Yaskawa INFORM job: DEMO_ROOF_UPPER_0625_3PAINT_4.JBI

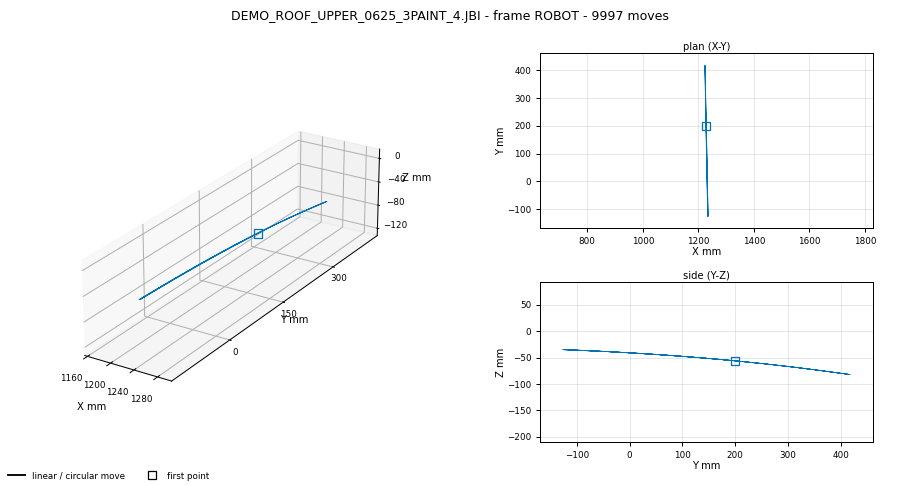
[picture p0: tool path of DEMO_ROOF_UPPER_0625_3PAINT_4.JBI in frame ROBOT, 9997 of 9997 moves have a stored position in this frame; points joined in program order, loops and branches not executed]
/JOB
//NAME DEMO_ROOF_UPPER_0625_3PAINT4
//POS
///NPOS 9997,0,0,0,0,0
///TOOL 0
///USER 0
///POSTYPE ROBOT
///RECTAN
///RCONF 1,0,0,0,0,0,0,0,0,0,0,0,0,0,0,0,0,0,0,0,0,0,0,0
C00000=1228.905,199.676,-56.077,-177.389,5.994,148.293
C00001=1228.909,199.428,-56.053,-177.392,5.993,148.294
C00002=1228.914,199.179,-56.029,-177.394,5.992,148.294
C00003=1228.919,198.930,-56.005,-177.396,5.990,148.294
C00004=1228.923,198.681,-55.981,-177.400,5.988,148.295
C00005=1228.928,198.432,-55.958,-177.402,5.986,148.295
C00006=1228.933,198.184,-55.934,-177.404,5.985,148.296
C00007=1228.937,197.935,-55.911,-177.407,5.983,148.296
C00008=1228.942,197.686,-55.887,-177.410,5.982,148.296
C00009=1228.946,197.437,-55.863,-177.412,5.980,148.297
C00010=1228.951,197.188,-55.840,-177.414,5.979,148.297
C00011=1228.956,196.939,-55.816,-177.417,5.977,148.298
C00012=1228.960,196.691,-55.792,-177.420,5.975,148.298
C00013=1228.965,196.442,-55.769,-177.423,5.973,148.298
C00014=1228.970,196.193,-55.746,-177.425,5.972,148.299
C00015=1228.974,195.944,-55.722,-177.427,5.971,148.299
C00016=1228.979,195.695,-55.698,-177.430,5.969,148.299
C00017=1228.983,195.446,-55.675,-177.433,5.968,148.300
C00018=1228.988,195.197,-55.652,-177.435,5.966,148.300
C00019=1228.992,194.949,-55.627,-177.438,5.964,148.301
C00020=1228.996,194.700,-55.605,-177.441,5.963,148.301
C00021=1229.001,194.451,-55.581,-177.443,5.961,148.301
C00022=1229.006,194.202,-55.558,-177.445,5.960,148.302
C00023=1229.010,193.953,-55.534,-177.448,5.958,148.302
C00024=1229.015,193.704,-55.511,-177.450,5.957,148.303
C00025=1229.020,193.455,-55.487,-177.453,5.955,148.303
C00026=1229.024,193.206,-55.464,-177.456,5.953,148.303
C00027=1229.029,192.957,-55.440,-177.458,5.952,148.304
C00028=1229.034,192.708,-55.417,-177.460,5.951,148.304
C00029=1229.039,192.461,-55.393,-177.464,5.949,148.305
C00030=1229.043,192.212,-55.371,-177.466,5.947,148.305
C00031=1229.047,191.963,-55.347,-177.468,5.946,148.305
C00032=1229.052,191.714,-55.324,-177.471,5.944,148.306
C00033=1229.057,191.465,-55.301,-177.474,5.942,148.306
C00034=1229.061,191.216,-55.277,-177.476,5.941,148.307
C00035=1229.066,190.967,-55.254,-177.479,5.940,148.307
C00036=1229.071,190.718,-55.231,-177.481,5.938,148.307
C00037=1229.075,190.469,-55.208,-177.484,5.937,148.308
C00038=1229.080,190.220,-55.184,-177.486,5.935,148.308
C00039=1229.084,189.971,-55.161,-177.489,5.933,148.308
C00040=1229.090,189.723,-55.138,-177.491,5.933,148.309
C00041=1229.094,189.474,-55.115,-177.494,5.931,148.309
C00042=1229.098,189.225,-55.092,-177.497,5.929,148.310
C00043=1229.103,188.976,-55.069,-177.499,5.928,148.310
C00044=1229.108,188.727,-55.045,-177.501,5.926,148.311
C00045=1229.112,188.478,-55.022,-177.505,5.925,148.311
C00046=1229.116,188.229,-54.999,-177.507,5.924,148.311
C00047=1229.121,187.980,-54.976,-177.509,5.922,148.312
C00048=1229.126,187.732,-54.953,-177.512,5.920,148.312
C00049=1229.131,187.483,-54.929,-177.514,5.919,148.313
C00050=1229.135,187.234,-54.907,-177.517,5.917,148.313
C00051=1229.140,186.985,-54.883,-177.520,5.916,148.313
C00052=1229.144,186.736,-54.860,-177.522,5.915,148.314
C00053=1229.149,186.487,-54.837,-177.525,5.913,148.314
C00054=1229.153,186.238,-54.814,-177.527,5.911,148.315
C00055=1229.158,185.968,-54.789,-177.530,5.909,148.315
C00056=1229.164,185.699,-54.764,-177.533,5.907,148.315
C00057=1229.168,185.429,-54.739,-177.536,5.907,148.316
C00058=1229.174,185.159,-54.714,-177.538,5.905,148.316
C00059=1229.178,184.910,-54.691,-177.541,5.903,148.317
C00060=1229.183,184.662,-54.668,-177.544,5.902,148.317
C00061=1229.187,184.413,-54.645,-177.546,5.901,148.318
C00062=1229.192,184.164,-54.622,-177.549,5.899,148.318
C00063=1229.196,183.915,-54.600,-177.551,5.898,148.318
C00064=1229.201,183.666,-54.576,-177.553,5.896,148.319
C00065=1229.206,183.418,-54.554,-177.557,5.894,148.319
C00066=1229.211,183.168,-54.531,-177.559,5.893,148.320
C00067=1229.215,182.919,-54.508,-177.561,5.892,148.320
C00068=1229.219,182.670,-54.485,-177.564,5.890,148.320
C00069=1229.225,182.422,-54.462,-177.567,5.889,148.321
C00070=1229.229,182.173,-54.440,-177.569,5.887,148.321
C00071=1229.234,181.924,-54.417,-177.572,5.885,148.322
C00072=1229.238,181.675,-54.393,-177.574,5.884,148.322
C00073=1229.242,181.426,-54.371,-177.577,5.883,148.323
C00074=1229.248,181.177,-54.348,-177.579,5.882,148.323
C00075=1229.252,180.928,-54.326,-177.582,5.880,148.323
C00076=1229.257,180.679,-54.302,-177.584,5.878,148.324
C00077=1229.261,180.431,-54.281,-177.587,5.877,148.324
C00078=1229.266,180.182,-54.257,-177.590,5.876,148.325
C00079=1229.270,179.932,-54.235,-177.592,5.874,148.325
C00080=1229.275,179.683,-54.212,-177.594,5.873,148.326
C00081=1229.280,179.435,-54.189,-177.598,5.871,148.326
C00082=1229.285,179.186,-54.167,-177.600,5.870,148.327
C00083=1229.289,178.936,-54.143,-177.602,5.868,148.327
C00084=1229.294,178.687,-54.121,-177.605,5.867,148.327
C00085=1229.299,178.439,-54.098,-177.608,5.866,148.328
C00086=1229.303,178.190,-54.076,-177.610,5.864,148.328
C00087=1229.307,177.941,-54.054,-177.612,5.863,148.329
C00088=1229.312,177.692,-54.031,-177.615,5.861,148.329
C00089=1229.317,177.443,-54.008,-177.618,5.860,148.329
C00090=1229.321,177.194,-53.985,-177.620,5.859,148.330
C00091=1229.326,176.945,-53.963,-177.623,5.857,148.330
C00092=1229.331,176.696,-53.940,-177.625,5.856,148.331
C00093=1229.335,176.447,-53.918,-177.628,5.854,148.331
C00094=1229.341,176.199,-53.895,-177.631,5.852,148.332
C00095=1229.345,175.949,-53.873,-177.633,5.851,148.332
C00096=1229.349,175.701,-53.850,-177.636,5.850,148.333
C00097=1229.354,175.452,-53.828,-177.638,5.849,148.333
C00098=1229.359,175.202,-53.806,-177.641,5.847,148.333
C00099=1229.363,174.953,-53.783,-177.643,5.845,148.334
C00100=1229.368,174.705,-53.761,-177.646,5.845,148.334
C00101=1229.372,174.456,-53.738,-177.649,5.843,148.335
C00102=1229.378,174.207,-53.716,-177.651,5.842,148.335
C00103=1229.382,173.958,-53.693,-177.654,5.840,148.336
C00104=1229.387,173.709,-53.670,-177.656,5.839,148.336
C00105=1229.392,173.460,-53.649,-177.658,5.837,148.336
C00106=1229.396,173.211,-53.626,-177.661,5.836,148.337
C00107=1229.401,172.962,-53.603,-177.664,5.835,148.337
C00108=1229.405,172.713,-53.582,-177.666,5.833,148.338
C00109=1229.409,172.464,-53.559,-177.668,5.832,148.338
C00110=1229.415,172.215,-53.537,-177.672,5.831,148.339
C00111=1229.419,171.966,-53.515,-177.674,5.830,148.339
C00112=1229.424,171.718,-53.492,-177.676,5.828,148.339
C00113=1229.428,171.469,-53.470,-177.679,5.826,148.340
C00114=1229.433,171.219,-53.447,-177.682,5.825,148.340
C00115=1229.438,170.970,-53.426,-177.684,5.823,148.341
C00116=1229.442,170.722,-53.403,-177.686,5.822,148.341
C00117=1229.448,170.473,-53.381,-177.689,5.821,148.342
C00118=1229.452,170.223,-53.359,-177.692,5.820,148.342
C00119=1229.457,169.975,-53.337,-177.694,5.818,148.342
C00120=1229.461,169.726,-53.314,-177.697,5.817,148.343
C00121=1229.466,169.476,-53.292,-177.699,5.816,148.343
C00122=1229.471,169.228,-53.270,-177.702,5.814,148.344
C00123=1229.475,168.978,-53.248,-177.705,5.813,148.344
C00124=1229.480,168.730,-53.226,-177.707,5.811,148.345
C00125=1229.485,168.480,-53.204,-177.709,5.810,148.345
C00126=1229.489,168.232,-53.181,-177.713,5.809,148.346
C00127=1229.494,167.983,-53.159,-177.715,5.808,148.346
C00128=1229.498,167.734,-53.137,-177.717,5.806,148.346
C00129=1229.503,167.485,-53.115,-177.720,5.805,148.347
C00130=1229.508,167.236,-53.093,-177.723,5.803,148.347
C00131=1229.513,166.986,-53.071,-177.725,5.802,148.348
C00132=1229.517,166.738,-53.049,-177.728,5.801,148.348
C00133=1229.522,166.488,-53.027,-177.730,5.800,148.349
C00134=1229.526,166.240,-53.005,-177.733,5.798,148.349
C00135=1229.531,165.991,-52.983,-177.736,5.797,148.350
C00136=1229.536,165.742,-52.961,-177.738,5.796,148.350
C00137=1229.540,165.493,-52.939,-177.740,5.794,148.350
C00138=1229.545,165.244,-52.917,-177.743,5.793,148.351
C00139=1229.550,164.995,-52.895,-177.746,5.791,148.351
C00140=1229.554,164.746,-52.873,-177.748,5.790,148.352
C00141=1229.559,164.497,-52.851,-177.751,5.789,148.352
C00142=1229.564,164.248,-52.829,-177.753,5.788,148.353
C00143=1229.568,163.999,-52.807,-177.756,5.786,148.353
C00144=1229.573,163.750,-52.786,-177.758,5.785,148.354
C00145=1229.578,163.501,-52.763,-177.761,5.783,148.354
C00146=1229.583,163.252,-52.741,-177.763,5.782,148.355
C00147=1229.587,163.003,-52.720,-177.766,5.781,148.355
C00148=1229.592,162.754,-52.698,-177.768,5.780,148.356
C00149=1229.597,162.505,-52.676,-177.771,5.778,148.356
C00150=1229.601,162.256,-52.654,-177.774,5.777,148.357
C00151=1229.606,162.007,-52.633,-177.776,5.776,148.357
C00152=1229.611,161.758,-52.611,-177.779,5.775,148.358
C00153=1229.615,161.509,-52.589,-177.781,5.773,148.358
C00154=1229.620,161.260,-52.568,-177.784,5.772,148.358
C00155=1229.624,161.011,-52.545,-177.787,5.771,148.359
C00156=1229.629,160.762,-52.524,-177.789,5.770,148.359
C00157=1229.634,160.513,-52.502,-177.791,5.768,148.360
C00158=1229.638,160.264,-52.480,-177.794,5.767,148.360
C00159=1229.644,159.995,-52.457,-177.797,5.765,148.361
C00160=1229.649,159.726,-52.434,-177.800,5.764,148.361
C00161=1229.654,159.457,-52.410,-177.802,5.763,148.362
C00162=1229.659,159.188,-52.386,-177.805,5.761,148.362
C00163=1229.663,158.938,-52.364,-177.807,5.760,148.363
C00164=1229.668,158.690,-52.343,-177.810,5.759,148.363
C00165=1229.673,158.441,-52.322,-177.812,5.758,148.364
C00166=1229.677,158.191,-52.300,-177.816,5.756,148.364
C00167=1229.682,157.943,-52.279,-177.818,5.755,148.365
C00168=1229.687,157.694,-52.257,-177.820,5.753,148.365
C00169=1229.691,157.444,-52.236,-177.823,5.753,148.366
C00170=1229.696,157.195,-52.214,-177.826,5.751,148.366
C00171=1229.701,156.947,-52.192,-177.828,5.750,148.366
C00172=1229.706,156.697,-52.171,-177.831,5.749,148.367
C00173=1229.711,156.448,-52.149,-177.833,5.748,148.367
C00174=1229.715,156.200,-52.128,-177.836,5.746,148.368
C00175=1229.720,155.950,-52.106,-177.838,5.745,148.368
C00176=1229.725,155.701,-52.085,-177.841,5.743,148.369
C00177=1229.729,155.453,-52.063,-177.843,5.743,148.369
C00178=1229.734,155.203,-52.042,-177.846,5.741,148.370
C00179=1229.738,154.954,-52.020,-177.849,5.740,148.370
C00180=1229.743,154.705,-51.999,-177.851,5.739,148.371
C00181=1229.748,154.456,-51.978,-177.853,5.737,148.371
C00182=1229.753,154.207,-51.956,-177.856,5.737,148.372
C00183=1229.757,153.958,-51.935,-177.859,5.735,148.372
C00184=1229.762,153.709,-51.914,-177.861,5.734,148.373
C00185=1229.766,153.460,-51.892,-177.864,5.732,148.373
C00186=1229.771,153.211,-51.871,-177.866,5.731,148.373
C00187=1229.776,152.962,-51.849,-177.869,5.730,148.374
C00188=1229.782,152.713,-51.828,-177.871,5.729,148.374
C00189=1229.785,152.464,-51.807,-177.874,5.727,148.375
C00190=1229.790,152.214,-51.786,-177.877,5.726,148.375
C00191=1229.795,151.966,-51.764,-177.879,5.726,148.376
C00192=1229.800,151.716,-51.743,-177.882,5.724,148.376
C00193=1229.804,151.467,-51.722,-177.884,5.723,148.377
C00194=1229.809,151.218,-51.701,-177.887,5.721,148.377
C00195=1229.814,150.970,-51.679,-177.889,5.720,148.378
C00196=1229.819,150.720,-51.658,-177.892,5.719,148.378
C00197=1229.823,150.471,-51.636,-177.894,5.718,148.379
C00198=1229.828,150.222,-51.615,-177.897,5.717,148.379
C00199=1229.833,149.973,-51.594,-177.900,5.715,148.380
C00200=1229.838,149.724,-51.573,-177.902,5.714,148.380
C00201=1229.842,149.476,-51.552,-177.905,5.713,148.381
C00202=1229.846,149.226,-51.530,-177.907,5.712,148.381
C00203=1229.852,148.977,-51.509,-177.910,5.710,148.382
C00204=1229.856,148.728,-51.488,-177.912,5.710,148.382
C00205=1229.861,148.479,-51.467,-177.915,5.709,148.383
C00206=1229.866,148.230,-51.446,-177.918,5.707,148.383
C00207=1229.870,147.980,-51.424,-177.920,5.706,148.384
C00208=1229.875,147.731,-51.404,-177.923,5.705,148.384
C00209=1229.880,147.483,-51.382,-177.925,5.704,148.385
C00210=1229.885,147.233,-51.361,-177.928,5.702,148.385
C00211=1229.889,146.985,-51.341,-177.930,5.701,148.386
C00212=1229.894,146.736,-51.319,-177.933,5.700,148.386
C00213=1229.898,146.486,-51.299,-177.935,5.699,148.387
C00214=1229.903,146.237,-51.278,-177.938,5.698,148.387
C00215=1229.908,145.988,-51.256,-177.941,5.696,148.388
C00216=1229.912,145.739,-51.236,-177.943,5.695,148.388
C00217=1229.918,145.490,-51.215,-177.945,5.695,148.389
C00218=1229.923,145.241,-51.194,-177.948,5.693,148.389
C00219=1229.926,144.992,-51.172,-177.951,5.692,148.390
C00220=1229.932,144.743,-51.151,-177.953,5.690,148.390
C00221=1229.936,144.494,-51.131,-177.956,5.690,148.391
C00222=1229.941,144.244,-51.110,-177.958,5.689,148.391
C00223=1229.945,143.996,-51.089,-177.961,5.687,148.392
C00224=1229.950,143.747,-51.068,-177.963,5.686,148.392
C00225=1229.956,143.498,-51.047,-177.967,5.685,148.393
C00226=1229.960,143.249,-51.026,-177.969,5.684,148.393
C00227=1229.965,142.999,-51.005,-177.971,5.683,148.394
C00228=1229.969,142.750,-50.985,-177.974,5.681,148.394
C00229=1229.974,142.501,-50.963,-177.976,5.681,148.395
C00230=1229.978,142.252,-50.943,-177.979,5.680,148.395
C00231=1229.984,142.003,-50.922,-177.981,5.678,148.395
C00232=1229.988,141.754,-50.901,-177.984,5.677,148.396
C00233=1229.993,141.505,-50.880,-177.987,5.675,148.396
C00234=1229.998,141.256,-50.860,-177.989,5.675,148.397
C00235=1230.003,141.006,-50.839,-177.991,5.674,148.397
C00236=1230.007,140.757,-50.819,-177.994,5.672,148.398
C00237=1230.012,140.509,-50.797,-177.997,5.671,148.398
C00238=1230.017,140.260,-50.777,-177.999,5.671,148.399
C00239=1230.021,140.010,-50.755,-178.002,5.669,148.399
C00240=1230.026,139.761,-50.735,-178.004,5.668,148.400
C00241=1230.031,139.512,-50.714,-178.007,5.666,148.400
C00242=1230.035,139.263,-50.694,-178.010,5.666,148.401
C00243=1230.040,139.014,-50.673,-178.012,5.665,148.401
C00244=1230.045,138.765,-50.652,-178.015,5.663,148.402
C00245=1230.049,138.516,-50.632,-178.017,5.662,148.403
C00246=1230.054,138.266,-50.611,-178.020,5.662,148.403
C00247=1230.059,138.017,-50.591,-178.022,5.660,148.404
C00248=1230.064,137.768,-50.570,-178.025,5.659,148.404
C00249=1230.068,137.519,-50.549,-178.027,5.658,148.405
C00250=1230.073,137.270,-50.529,-178.030,5.657,148.405
C00251=1230.078,137.021,-50.508,-178.032,5.656,148.406
C00252=1230.082,136.772,-50.487,-178.035,5.654,148.406
C00253=1230.087,136.523,-50.467,-178.038,5.653,148.407
C00254=1230.092,136.273,-50.447,-178.040,5.653,148.407
C00255=1230.097,136.024,-50.426,-178.043,5.651,148.408
C00256=1230.102,135.775,-50.406,-178.045,5.650,148.408
C00257=1230.106,135.526,-50.385,-178.048,5.649,148.409
C00258=1230.111,135.277,-50.365,-178.051,5.648,148.409
C00259=1230.116,135.028,-50.344,-178.053,5.647,148.410
C00260=1230.121,134.779,-50.323,-178.055,5.646,148.410
C00261=1230.125,134.530,-50.303,-178.058,5.644,148.411
C00262=1230.130,134.280,-50.283,-178.061,5.644,148.411
C00263=1230.135,134.012,-50.261,-178.063,5.643,148.412
C00264=1230.140,133.744,-50.239,-178.066,5.641,148.412
C00265=1230.146,133.475,-50.217,-178.069,5.640,148.413
C00266=1230.150,133.206,-50.195,-178.072,5.639,148.414
C00267=1230.155,132.957,-50.174,-178.074,5.638,148.414
C00268=1230.160,132.707,-50.154,-178.077,5.637,148.415
C00269=1230.165,132.459,-50.134,-178.079,5.636,148.415
C00270=1230.170,132.210,-50.113,-178.082,5.635,148.416
C00271=1230.175,131.961,-50.093,-178.084,5.633,148.416
C00272=1230.179,131.711,-50.073,-178.087,5.632,148.417
C00273=1230.184,131.462,-50.053,-178.089,5.631,148.417
C00274=1230.189,131.213,-50.032,-178.092,5.630,148.418
C00275=1230.193,130.964,-50.011,-178.095,5.629,148.418
C00276=1230.198,130.714,-49.992,-178.097,5.628,148.419
C00277=1230.203,130.465,-49.971,-178.100,5.627,148.419
C00278=1230.207,130.217,-49.951,-178.102,5.626,148.420
C00279=1230.212,129.967,-49.931,-178.105,5.625,148.420
C00280=1230.218,129.718,-49.911,-178.107,5.624,148.421
C00281=1230.222,129.469,-49.890,-178.110,5.623,148.421
C00282=1230.227,129.220,-49.871,-178.112,5.622,148.422
C00283=1230.231,128.971,-49.850,-178.115,5.621,148.422
C00284=1230.236,128.722,-49.829,-178.118,5.619,148.423
C00285=1230.241,128.472,-49.810,-178.120,5.619,148.423
C00286=1230.246,128.223,-49.789,-178.123,5.618,148.424
C00287=1230.250,127.974,-49.770,-178.125,5.616,148.424
C00288=1230.255,127.725,-49.750,-178.128,5.616,148.425
C00289=1230.260,127.476,-49.729,-178.130,5.615,148.425
C00290=1230.265,127.226,-49.709,-178.133,5.613,148.426
C00291=1230.270,126.978,-49.689,-178.135,5.612,148.426
C00292=1230.274,126.728,-49.669,-178.138,5.612,148.427
C00293=1230.279,126.479,-49.649,-178.140,5.611,148.428
C00294=1230.284,126.230,-49.629,-178.143,5.609,148.428
C00295=1230.289,125.981,-49.609,-178.146,5.609,148.429
C00296=1230.293,125.732,-49.589,-178.148,5.608,148.429
C00297=1230.298,125.483,-49.569,-178.151,5.606,148.430
C00298=1230.302,125.234,-49.549,-178.153,5.605,148.430
C00299=1230.307,124.984,-49.529,-178.156,5.605,148.431
C00300=1230.313,124.736,-49.508,-178.158,5.604,148.431
C00301=1230.317,124.486,-49.489,-178.161,5.602,148.432
C00302=1230.322,124.236,-49.469,-178.164,5.601,148.432
C00303=1230.327,123.988,-49.449,-178.166,5.600,148.433
C00304=1230.331,123.738,-49.429,-178.169,5.599,148.434
C00305=1230.336,123.490,-49.409,-178.171,5.598,148.434
C00306=1230.341,123.240,-49.389,-178.174,5.597,148.435
C00307=1230.346,122.991,-49.369,-178.176,5.596,148.435
C00308=1230.350,122.742,-49.349,-178.179,5.595,148.436
C00309=1230.355,122.493,-49.329,-178.182,5.594,148.436
C00310=1230.360,122.244,-49.310,-178.184,5.593,148.437
C00311=1230.365,121.994,-49.290,-178.186,5.593,148.437
C00312=1230.369,121.745,-49.270,-178.189,5.591,148.438
C00313=1230.374,121.496,-49.250,-178.192,5.590,148.438
C00314=1230.379,121.247,-49.231,-178.194,5.590,148.439
C00315=1230.384,120.998,-49.210,-178.196,5.589,148.439
C00316=1230.389,120.748,-49.191,-178.200,5.587,148.440
C00317=1230.393,120.499,-49.171,-178.202,5.586,148.440
C00318=1230.398,120.251,-49.151,-178.204,5.586,148.441
C00319=1230.403,120.001,-49.131,-178.206,5.585,148.441
C00320=1230.408,119.751,-49.112,-178.210,5.583,148.442
C00321=1230.413,119.503,-49.092,-178.212,5.583,148.443
C00322=1230.418,119.254,-49.072,-178.214,5.582,148.443
C00323=1230.422,119.004,-49.053,-178.217,5.581,148.444
C00324=1230.426,118.755,-49.033,-178.220,5.579,148.444
C00325=1230.431,118.507,-49.013,-178.222,5.579,148.445
C00326=1230.436,118.257,-48.994,-178.225,5.578,148.445
C00327=1230.441,118.007,-48.974,-178.227,5.577,148.446
C00328=1230.446,117.759,-48.955,-178.230,5.575,148.446
C00329=1230.451,117.510,-48.934,-178.233,5.575,148.447
C00330=1230.455,117.260,-48.915,-178.235,5.574,148.447
C00331=1230.461,117.011,-48.895,-178.237,5.573,148.448
C00332=1230.466,116.762,-48.876,-178.240,5.571,148.449
C00333=1230.470,116.512,-48.857,-178.243,5.571,148.449
C00334=1230.474,116.263,-48.836,-178.245,5.570,148.450
C00335=1230.479,116.014,-48.817,-178.247,5.569,148.450
C00336=1230.484,115.765,-48.797,-178.251,5.568,148.451
C00337=1230.489,115.516,-48.778,-178.253,5.567,148.451
C00338=1230.494,115.266,-48.758,-178.255,5.566,148.452
C00339=1230.499,115.017,-48.739,-178.258,5.566,148.453
C00340=1230.503,114.768,-48.720,-178.261,5.564,148.453
C00341=1230.508,114.519,-48.700,-178.263,5.563,148.454
C00342=1230.513,114.270,-48.680,-178.266,5.563,148.454
C00343=1230.518,114.021,-48.661,-178.268,5.562,148.455
C00344=1230.523,113.771,-48.641,-178.271,5.561,148.455
C00345=1230.527,113.522,-48.622,-178.273,5.559,148.456
C00346=1230.532,113.273,-48.603,-178.276,5.559,148.456
C00347=1230.537,113.024,-48.583,-178.279,5.558,148.457
C00348=1230.542,112.775,-48.564,-178.281,5.557,148.457
C00349=1230.547,112.525,-48.544,-178.283,5.556,148.458
C00350=1230.551,112.276,-48.525,-178.286,5.555,148.459
C00351=1230.556,112.027,-48.506,-178.289,5.554,148.459
C00352=1230.561,111.778,-48.486,-178.291,5.553,148.460
C00353=1230.566,111.529,-48.467,-178.293,5.552,148.460
C00354=1230.570,111.279,-48.448,-178.296,5.551,148.461
C00355=1230.575,111.030,-48.428,-178.299,5.550,148.461
C00356=1230.580,110.781,-48.409,-178.301,5.549,148.462
C00357=1230.584,110.532,-48.390,-178.304,5.549,148.462
C00358=1230.590,110.283,-48.370,-178.306,5.548,148.463
C00359=1230.595,110.033,-48.351,-178.309,5.546,148.463
C00360=1230.599,109.784,-48.331,-178.312,5.546,148.464
C00361=1230.604,109.535,-48.312,-178.314,5.545,148.465
C00362=1230.609,109.286,-48.293,-178.316,5.544,148.465
C00363=1230.614,109.037,-48.274,-178.319,5.543,148.466
C00364=1230.618,108.788,-48.254,-178.322,5.542,148.466
C00365=1230.623,108.539,-48.235,-178.324,5.541,148.467
C00366=1230.628,108.288,-48.216,-178.327,5.540,148.467
C00367=1230.633,108.021,-48.196,-178.330,5.540,148.468
C00368=1230.638,107.752,-48.175,-178.333,5.538,148.469
C00369=1230.643,107.484,-48.154,-178.335,5.537,148.469
C00370=1230.649,107.215,-48.134,-178.338,5.537,148.470
C00371=1230.654,106.965,-48.114,-178.341,5.535,148.470
C00372=1230.658,106.717,-48.096,-178.343,5.535,148.471
C00373=1230.663,106.467,-48.076,-178.345,5.534,148.472
C00374=1230.668,106.218,-48.057,-178.348,5.533,148.472
C00375=1230.673,105.969,-48.038,-178.351,5.532,148.473
C00376=1230.678,105.720,-48.019,-178.353,5.531,148.473
C00377=1230.682,105.470,-48.000,-178.356,5.530,148.474
C00378=1230.687,105.222,-47.981,-178.359,5.529,148.474
C00379=1230.691,104.972,-47.962,-178.361,5.528,148.475
C00380=1230.697,104.723,-47.943,-178.363,5.528,148.476
C00381=1230.702,104.473,-47.923,-178.366,5.527,148.476
C00382=1230.706,104.225,-47.905,-178.368,5.526,148.477
C00383=1230.711,103.975,-47.885,-178.371,5.525,148.477
C00384=1230.716,103.726,-47.867,-178.374,5.524,148.478
C00385=1230.721,103.476,-47.847,-178.376,5.523,148.478
C00386=1230.725,103.228,-47.829,-178.379,5.523,148.479
C00387=1230.731,102.978,-47.810,-178.381,5.522,148.480
C00388=1230.735,102.729,-47.791,-178.383,5.521,148.480
C00389=1230.740,102.480,-47.772,-178.386,5.520,148.481
C00390=1230.745,102.230,-47.753,-178.389,5.519,148.481
C00391=1230.750,101.981,-47.734,-178.392,5.518,148.482
C00392=1230.754,101.732,-47.715,-178.394,5.517,148.482
C00393=1230.760,101.483,-47.696,-178.396,5.517,148.483
C00394=1230.764,101.233,-47.677,-178.399,5.516,148.484
C00395=1230.769,100.985,-47.658,-178.402,5.514,148.484
C00396=1230.774,100.735,-47.640,-178.404,5.514,148.485
C00397=1230.779,100.486,-47.620,-178.407,5.513,148.485
C00398=1230.783,100.237,-47.603,-178.409,5.512,148.486
C00399=1230.788,99.987,-47.583,-178.412,5.512,148.486
C00400=1230.793,99.739,-47.564,-178.414,5.511,148.487
C00401=1230.798,99.488,-47.545,-178.416,5.510,148.487
C00402=1230.802,99.240,-47.527,-178.420,5.509,148.488
C00403=1230.807,98.991,-47.509,-178.422,5.508,148.489
C00404=1230.812,98.741,-47.489,-178.425,5.507,148.489
C00405=1230.817,98.492,-47.471,-178.427,5.506,148.490
C00406=1230.822,98.243,-47.452,-178.430,5.506,148.490
C00407=1230.827,97.993,-47.433,-178.432,5.505,148.491
C00408=1230.832,97.744,-47.414,-178.434,5.504,148.492
C00409=1230.836,97.494,-47.396,-178.437,5.504,148.492
C00410=1230.841,97.246,-47.377,-178.440,5.502,148.493
C00411=1230.847,96.996,-47.358,-178.442,5.501,148.493
C00412=1230.851,96.747,-47.339,-178.445,5.501,148.494
C00413=1230.856,96.498,-47.321,-178.448,5.500,148.495
C00414=1230.861,96.249,-47.302,-178.450,5.499,148.495
C00415=1230.865,95.999,-47.284,-178.452,5.498,148.496
C00416=1230.871,95.750,-47.264,-178.455,5.498,148.496
C00417=1230.875,95.501,-47.246,-178.458,5.497,148.497
C00418=1230.880,95.251,-47.228,-178.460,5.495,148.497
C00419=1230.885,95.002,-47.209,-178.463,5.495,148.498
C00420=1230.890,94.753,-47.191,-178.465,5.494,148.499
C00421=1230.894,94.504,-47.172,-178.468,5.494,148.499
C00422=1230.900,94.254,-47.153,-178.470,5.493,148.500
C00423=1230.905,94.005,-47.135,-178.473,5.492,148.500
C00424=1230.909,93.756,-47.116,-178.475,5.491,148.501
C00425=1230.914,93.507,-47.098,-178.478,5.491,148.502
C00426=1230.919,93.257,-47.080,-178.481,5.489,148.502
C00427=1230.923,93.008,-47.061,-178.483,5.488,148.503
C00428=1230.928,92.759,-47.043,-178.486,5.488,148.503
C00429=1230.934,92.509,-47.024,-178.488,5.487,148.504
C00430=1230.938,92.260,-47.005,-178.491,5.486,148.504
C00431=1230.943,92.011,-46.987,-178.493,5.486,148.505
C00432=1230.948,91.762,-46.969,-178.496,5.485,148.506
C00433=1230.953,91.513,-46.950,-178.498,5.484,148.506
C00434=1230.957,91.263,-46.931,-178.501,5.483,148.507
C00435=1230.962,91.014,-46.913,-178.503,5.483,148.507
C00436=1230.967,90.765,-46.895,-178.507,5.481,148.508
C00437=1230.971,90.515,-46.876,-178.509,5.480,148.509
C00438=1230.977,90.266,-46.858,-178.511,5.480,148.509
C00439=1230.982,90.017,-46.840,-178.514,5.479,148.510
C00440=1230.987,89.768,-46.822,-178.517,5.479,148.510
C00441=1230.991,89.518,-46.803,-178.519,5.478,148.511
C00442=1230.996,89.269,-46.784,-178.521,5.477,148.512
C00443=1231.001,89.020,-46.766,-178.524,5.476,148.512
C00444=1231.006,88.771,-46.748,-178.527,5.476,148.513
C00445=1231.010,88.521,-46.730,-178.529,5.475,148.513
C00446=1231.015,88.272,-46.711,-178.531,5.474,148.514
C00447=1231.020,88.023,-46.693,-178.534,5.473,148.515
C00448=1231.025,87.773,-46.675,-178.537,5.472,148.515
C00449=1231.030,87.524,-46.657,-178.539,5.471,148.516
C00450=1231.035,87.274,-46.638,-178.542,5.471,148.516
C00451=1231.040,87.025,-46.620,-178.544,5.470,148.517
C00452=1231.045,86.776,-46.602,-178.547,5.469,148.518
C00453=1231.049,86.527,-46.584,-178.549,5.468,148.518
C00454=1231.054,86.278,-46.566,-178.552,5.468,148.519
C00455=1231.058,86.028,-46.547,-178.554,5.467,148.519
C00456=1231.064,85.779,-46.529,-178.557,5.467,148.520
C00457=1231.069,85.530,-46.511,-178.559,5.466,148.520
C00458=1231.074,85.281,-46.493,-178.562,5.465,148.521
C00459=1231.079,85.031,-46.475,-178.564,5.465,148.522
C00460=1231.083,84.782,-46.456,-178.568,5.463,148.522
C00461=1231.088,84.532,-46.438,-178.570,5.462,148.523
C00462=1231.093,84.283,-46.420,-178.572,5.462,148.523
C00463=1231.098,84.034,-46.402,-178.575,5.461,148.524
C00464=1231.103,83.785,-46.384,-178.578,5.460,148.525
C00465=1231.108,83.536,-46.366,-178.580,5.460,148.525
C00466=1231.112,83.286,-46.348,-178.582,5.459,148.526
C00467=1231.117,83.037,-46.330,-178.585,5.458,148.527
C00468=1231.122,82.787,-46.312,-178.588,5.458,148.527
C00469=1231.127,82.538,-46.294,-178.590,5.457,148.528
C00470=1231.132,82.289,-46.276,-178.592,5.456,148.528
C00471=1231.137,82.021,-46.256,-178.595,5.455,148.529
C00472=1231.142,81.752,-46.237,-178.598,5.454,148.530
C00473=1231.148,81.484,-46.217,-178.601,5.453,148.530
C00474=1231.153,81.215,-46.199,-178.603,5.453,148.531
C00475=1231.158,80.966,-46.181,-178.606,5.452,148.532
C00476=1231.163,80.717,-46.163,-178.609,5.452,148.532
C00477=1231.168,80.468,-46.145,-178.611,5.451,148.533
C00478=1231.172,80.218,-46.126,-178.614,5.450,148.533
C00479=1231.177,79.969,-46.108,-178.616,5.449,148.534
C00480=1231.182,79.719,-46.090,-178.619,5.449,148.535
C00481=1231.187,79.470,-46.072,-178.621,5.448,148.535
C00482=1231.192,79.221,-46.054,-178.624,5.448,148.536
C00483=1231.197,78.971,-46.037,-178.626,5.447,148.536
C00484=1231.202,78.722,-46.019,-178.629,5.446,148.537
C00485=1231.207,78.473,-46.001,-178.631,5.446,148.538
C00486=1231.211,78.224,-45.984,-178.634,5.445,148.538
C00487=1231.216,77.975,-45.966,-178.637,5.444,148.539
C00488=1231.221,77.725,-45.949,-178.639,5.443,148.539
C00489=1231.226,77.476,-45.931,-178.642,5.442,148.540
C00490=1231.230,77.226,-45.912,-178.645,5.441,148.541
C00491=1231.235,76.977,-45.894,-178.647,5.441,148.541
C00492=1231.240,76.728,-45.876,-178.650,5.440,148.542
C00493=1231.245,76.478,-45.859,-178.652,5.439,148.542
C00494=1231.250,76.229,-45.841,-178.655,5.439,148.543
C00495=1231.254,75.980,-45.824,-178.657,5.438,148.544
C00496=1231.259,75.731,-45.806,-178.660,5.437,148.544
C00497=1231.264,75.481,-45.788,-178.662,5.437,148.545
C00498=1231.269,75.232,-45.770,-178.665,5.436,148.545
C00499=1231.274,74.982,-45.753,-178.667,5.435,148.546
C00500=1231.279,74.733,-45.735,-178.670,5.435,148.547
C00501=1231.284,74.484,-45.717,-178.672,5.434,148.547
C00502=1231.289,74.235,-45.700,-178.675,5.434,148.548
C00503=1231.293,73.985,-45.682,-178.677,5.433,148.549
C00504=1231.299,73.736,-45.665,-178.680,5.432,148.549
C00505=1231.304,73.487,-45.647,-178.683,5.431,148.550
C00506=1231.309,73.237,-45.629,-178.685,5.431,148.551
C00507=1231.313,72.988,-45.612,-178.688,5.430,148.551
C00508=1231.318,72.739,-45.594,-178.690,5.430,148.552
C00509=1231.323,72.489,-45.577,-178.693,5.429,148.552
C00510=1231.328,72.240,-45.559,-178.695,5.428,148.553
C00511=1231.333,71.991,-45.541,-178.698,5.428,148.554
C00512=1231.337,71.741,-45.524,-178.700,5.427,148.554
C00513=1231.342,71.492,-45.506,-178.703,5.426,148.555
C00514=1231.348,71.242,-45.489,-178.705,5.425,148.555
C00515=1231.352,70.993,-45.471,-178.708,5.425,148.556
C00516=1231.357,70.744,-45.454,-178.710,5.424,148.557
C00517=1231.362,70.494,-45.436,-178.713,5.424,148.557
C00518=1231.367,70.245,-45.418,-178.716,5.423,148.558
C00519=1231.372,69.995,-45.401,-178.718,5.422,148.559
C00520=1231.376,69.746,-45.384,-178.720,5.422,148.559
C00521=1231.381,69.497,-45.366,-178.723,5.421,148.560
C00522=1231.387,69.248,-45.349,-178.726,5.420,148.560
C00523=1231.391,68.999,-45.332,-178.728,5.420,148.561
C00524=1231.396,68.749,-45.314,-178.731,5.419,148.562
C00525=1231.402,68.500,-45.297,-178.734,5.419,148.562
C00526=1231.406,68.250,-45.279,-178.736,5.418,148.563
C00527=1231.411,68.001,-45.262,-178.738,5.417,148.564
C00528=1231.416,67.752,-45.244,-178.741,5.416,148.564
C00529=1231.421,67.502,-45.227,-178.744,5.416,148.565
C00530=1231.425,67.253,-45.210,-178.746,5.415,148.565
C00531=1231.430,67.003,-45.192,-178.749,5.415,148.566
C00532=1231.436,66.754,-45.175,-178.751,5.414,148.567
C00533=1231.440,66.505,-45.158,-178.754,5.413,148.567
C00534=1231.446,66.256,-45.141,-178.756,5.413,148.568
C00535=1231.450,66.007,-45.123,-178.759,5.412,148.569
C00536=1231.455,65.757,-45.106,-178.762,5.411,148.569
C00537=1231.460,65.508,-45.088,-178.764,5.411,148.570
C00538=1231.464,65.258,-45.071,-178.767,5.410,148.571
C00539=1231.470,65.009,-45.054,-178.769,5.409,148.571
C00540=1231.475,64.759,-45.036,-178.772,5.409,148.572
C00541=1231.479,64.510,-45.020,-178.774,5.409,148.572
C00542=1231.485,64.261,-45.003,-178.776,5.408,148.573
C00543=1231.489,64.012,-44.985,-178.779,5.408,148.574
C00544=1231.494,63.762,-44.968,-178.782,5.407,148.574
C00545=1231.499,63.513,-44.951,-178.784,5.406,148.575
C00546=1231.504,63.263,-44.933,-178.786,5.406,148.575
C00547=1231.509,63.014,-44.916,-178.789,5.405,148.576
C00548=1231.513,62.764,-44.899,-178.792,5.404,148.577
C00549=1231.519,62.516,-44.882,-178.794,5.404,148.577
C00550=1231.523,62.266,-44.865,-178.797,5.403,148.578
C00551=1231.529,62.016,-44.848,-178.799,5.403,148.579
C00552=1231.533,61.767,-44.831,-178.802,5.402,148.579
C00553=1231.538,61.518,-44.813,-178.804,5.401,148.580
C00554=1231.542,61.268,-44.797,-178.807,5.401,148.581
C00555=1231.548,61.019,-44.780,-178.810,5.400,148.581
C00556=1231.553,60.770,-44.763,-178.812,5.399,148.582
C00557=1231.558,60.520,-44.746,-178.815,5.399,148.583
C00558=1231.562,60.271,-44.728,-178.817,5.398,148.583
C00559=1231.567,60.021,-44.711,-178.820,5.398,148.584
C00560=1231.572,59.772,-44.695,-178.822,5.397,148.584
C00561=1231.578,59.523,-44.678,-178.825,5.396,148.585
C00562=1231.582,59.273,-44.661,-178.827,5.396,148.586
C00563=1231.587,59.024,-44.643,-178.830,5.395,148.586
C00564=1231.592,58.775,-44.627,-178.832,5.395,148.587
C00565=1231.597,58.525,-44.609,-178.835,5.395,148.588
C00566=1231.602,58.276,-44.593,-178.837,5.394,148.588
C00567=1231.607,58.026,-44.575,-178.840,5.393,148.589
C00568=1231.612,57.777,-44.559,-178.842,5.393,148.589
C00569=1231.617,57.528,-44.542,-178.845,5.392,148.590
C00570=1231.621,57.279,-44.524,-178.847,5.391,148.591
C00571=1231.626,57.029,-44.508,-178.850,5.391,148.591
C00572=1231.631,56.779,-44.490,-178.853,5.390,148.592
C00573=1231.636,56.531,-44.474,-178.855,5.390,148.593
C00574=1231.641,56.281,-44.457,-178.858,5.389,148.593
C00575=1231.646,56.012,-44.439,-178.861,5.389,148.594
C00576=1231.652,55.744,-44.420,-178.863,5.388,148.595
C00577=1231.657,55.476,-44.402,-178.866,5.387,148.595
C00578=1231.662,55.208,-44.385,-178.869,5.387,148.596
C00579=1231.667,54.958,-44.367,-178.871,5.386,148.597
C00580=1231.672,54.708,-44.351,-178.874,5.386,148.597
C00581=1231.678,54.459,-44.334,-178.876,5.385,148.598
C00582=1231.682,54.210,-44.317,-178.879,5.385,148.599
C00583=1231.687,53.960,-44.300,-178.881,5.384,148.599
C00584=1231.692,53.711,-44.284,-178.884,5.383,148.600
C00585=1231.697,53.462,-44.267,-178.886,5.382,148.601
C00586=1231.701,53.212,-44.250,-178.889,5.383,148.601
C00587=1231.707,52.962,-44.233,-178.891,5.382,148.602
C00588=1231.712,52.714,-44.217,-178.894,5.382,148.603
C00589=1231.716,52.464,-44.201,-178.896,5.381,148.603
C00590=1231.722,52.214,-44.183,-178.899,5.380,148.604
C00591=1231.727,51.965,-44.167,-178.902,5.380,148.605
C00592=1231.731,51.716,-44.150,-178.904,5.379,148.605
C00593=1231.736,51.466,-44.134,-178.907,5.378,148.606
C00594=1231.741,51.217,-44.117,-178.909,5.378,148.606
C00595=1231.746,50.967,-44.100,-178.912,5.377,148.607
C00596=1231.750,50.718,-44.084,-178.914,5.377,148.608
C00597=1231.756,50.469,-44.067,-178.916,5.377,148.608
C00598=1231.761,50.219,-44.050,-178.919,5.376,148.609
C00599=1231.765,49.970,-44.033,-178.922,5.376,148.610
C00600=1231.771,49.721,-44.018,-178.924,5.375,148.610
C00601=1231.776,49.471,-44.000,-178.927,5.375,148.611
C00602=1231.781,49.222,-43.984,-178.929,5.374,148.611
C00603=1231.785,48.972,-43.968,-178.932,5.373,148.612
C00604=1231.790,48.723,-43.951,-178.934,5.372,148.613
C00605=1231.796,48.474,-43.934,-178.937,5.372,148.613
C00606=1231.800,48.224,-43.918,-178.940,5.371,148.614
C00607=1231.805,47.974,-43.901,-178.942,5.372,148.615
C00608=1231.810,47.726,-43.885,-178.944,5.371,148.615
C00609=1231.814,47.476,-43.868,-178.947,5.370,148.616
C00610=1231.820,47.227,-43.851,-178.950,5.370,148.617
C00611=1231.825,46.977,-43.835,-178.952,5.369,148.617
C00612=1231.830,46.727,-43.819,-178.955,5.369,148.618
C00613=1231.835,46.479,-43.803,-178.957,5.368,148.619
C00614=1231.839,46.229,-43.786,-178.960,5.367,148.619
C00615=1231.845,45.980,-43.770,-178.962,5.367,148.620
C00616=1231.850,45.730,-43.753,-178.964,5.367,148.621
C00617=1231.854,45.480,-43.736,-178.967,5.366,148.621
C00618=1231.860,45.231,-43.721,-178.970,5.366,148.622
C00619=1231.864,44.982,-43.704,-178.972,5.365,148.623
C00620=1231.869,44.733,-43.688,-178.975,5.365,148.623
C00621=1231.874,44.483,-43.671,-178.978,5.364,148.624
C00622=1231.879,44.234,-43.656,-178.980,5.364,148.625
C00623=1231.884,43.984,-43.638,-178.983,5.363,148.625
C00624=1231.889,43.735,-43.622,-178.985,5.363,148.626
C00625=1231.894,43.485,-43.606,-178.987,5.362,148.626
C00626=1231.899,43.236,-43.589,-178.990,5.362,148.627
C00627=1231.904,42.986,-43.574,-178.992,5.361,148.628
C00628=1231.908,42.737,-43.557,-178.995,5.361,148.628
C00629=1231.914,42.488,-43.541,-178.998,5.360,148.629
C00630=1231.918,42.238,-43.525,-179.000,5.359,148.630
C00631=1231.923,41.989,-43.509,-179.003,5.359,148.630
C00632=1231.928,41.740,-43.492,-179.005,5.359,148.631
C00633=1231.934,41.490,-43.476,-179.008,5.359,148.632
C00634=1231.938,41.240,-43.459,-179.010,5.358,148.633
C00635=1231.944,40.991,-43.443,-179.013,5.357,148.633
C00636=1231.948,40.742,-43.427,-179.016,5.357,148.634
C00637=1231.954,40.492,-43.411,-179.018,5.356,148.635
C00638=1231.958,40.243,-43.394,-179.021,5.356,148.635
C00639=1231.964,39.993,-43.379,-179.022,5.356,148.636
C00640=1231.968,39.744,-43.362,-179.025,5.355,148.636
C00641=1231.973,39.495,-43.346,-179.028,5.354,148.637
C00642=1231.978,39.245,-43.330,-179.030,5.354,148.638
C00643=1231.983,38.996,-43.314,-179.033,5.353,148.638
C00644=1231.988,38.746,-43.298,-179.036,5.353,148.639
C00645=1231.993,38.497,-43.281,-179.038,5.352,148.640
C00646=1231.998,38.247,-43.265,-179.040,5.352,148.640
C00647=1232.003,37.998,-43.250,-179.043,5.352,148.641
C00648=1232.008,37.748,-43.233,-179.046,5.351,148.642
C00649=1232.013,37.499,-43.218,-179.048,5.351,148.642
C00650=1232.017,37.249,-43.201,-179.051,5.350,148.643
C00651=1232.023,37.000,-43.185,-179.054,5.350,148.644
C00652=1232.028,36.751,-43.169,-179.056,5.349,148.644
C00653=1232.033,36.501,-43.153,-179.058,5.349,148.645
C00654=1232.038,36.252,-43.137,-179.061,5.349,148.646
C00655=1232.043,36.002,-43.121,-179.064,5.348,148.646
C00656=1232.048,35.753,-43.105,-179.066,5.347,148.647
C00657=1232.052,35.504,-43.089,-179.068,5.347,148.648
C00658=1232.057,35.254,-43.074,-179.071,5.346,148.648
C00659=1232.062,35.005,-43.057,-179.073,5.346,148.649
C00660=1232.067,34.755,-43.041,-179.076,5.346,148.650
C00661=1232.072,34.506,-43.026,-179.078,5.345,148.650
C00662=1232.077,34.256,-43.009,-179.081,5.345,148.651
C00663=1232.082,34.007,-42.993,-179.084,5.344,148.652
C00664=1232.087,33.757,-42.978,-179.086,5.344,148.652
C00665=1232.092,33.508,-42.961,-179.088,5.344,148.653
C00666=1232.097,33.259,-42.946,-179.091,5.343,148.654
C00667=1232.101,33.009,-42.930,-179.094,5.343,148.654
C00668=1232.107,32.760,-42.914,-179.096,5.342,148.655
C00669=1232.111,32.510,-42.898,-179.099,5.342,148.656
C00670=1232.117,32.261,-42.882,-179.102,5.341,148.656
C00671=1232.122,32.011,-42.867,-179.104,5.341,148.657
C00672=1232.127,31.762,-42.850,-179.106,5.341,148.658
C00673=1232.132,31.512,-42.835,-179.109,5.340,148.658
C00674=1232.137,31.263,-42.820,-179.112,5.340,148.659
C00675=1232.141,31.013,-42.804,-179.114,5.339,148.660
C00676=1232.147,30.764,-42.787,-179.117,5.339,148.660
C00677=1232.151,30.514,-42.771,-179.118,5.339,148.661
C00678=1232.157,30.265,-42.756,-179.121,5.338,148.662
C00679=1232.162,29.996,-42.739,-179.124,5.338,148.662
C00680=1232.167,29.728,-42.722,-179.127,5.337,148.663
C00681=1232.173,29.460,-42.705,-179.130,5.337,148.664
C00682=1232.178,29.191,-42.688,-179.132,5.336,148.665
C00683=1232.183,28.941,-42.672,-179.135,5.336,148.665
C00684=1232.188,28.692,-42.657,-179.137,5.335,148.666
C00685=1232.192,28.442,-42.641,-179.140,5.335,148.667
C00686=1232.197,28.193,-42.625,-179.142,5.335,148.667
C00687=1232.203,27.944,-42.610,-179.145,5.334,148.668
C00688=1232.208,27.694,-42.594,-179.147,5.334,148.669
C00689=1232.212,27.445,-42.579,-179.150,5.333,148.669
C00690=1232.218,27.195,-42.563,-179.153,5.332,148.670
C00691=1232.222,26.945,-42.547,-179.155,5.333,148.671
C00692=1232.228,26.696,-42.531,-179.157,5.332,148.671
C00693=1232.233,26.447,-42.516,-179.160,5.332,148.672
C00694=1232.238,26.198,-42.500,-179.163,5.331,148.673
C00695=1232.242,25.948,-42.484,-179.165,5.331,148.673
C00696=1232.247,25.699,-42.469,-179.167,5.331,148.674
C00697=1232.252,25.449,-42.454,-179.170,5.330,148.675
C00698=1232.257,25.199,-42.438,-179.173,5.330,148.675
C00699=1232.263,24.950,-42.422,-179.175,5.329,148.676
C00700=1232.267,24.701,-42.407,-179.178,5.329,148.677
C00701=1232.273,24.451,-42.391,-179.180,5.329,148.677
C00702=1232.277,24.201,-42.376,-179.183,5.328,148.678
C00703=1232.282,23.952,-42.361,-179.185,5.328,148.679
C00704=1232.287,23.703,-42.345,-179.188,5.327,148.679
C00705=1232.293,23.453,-42.329,-179.190,5.327,148.680
C00706=1232.297,23.203,-42.314,-179.193,5.327,148.681
C00707=1232.302,22.954,-42.298,-179.195,5.326,148.682
C00708=1232.307,22.705,-42.283,-179.198,5.326,148.682
C00709=1232.312,22.456,-42.268,-179.200,5.325,148.683
C00710=1232.317,22.205,-42.252,-179.202,5.325,148.683
C00711=1232.322,21.956,-42.237,-179.205,5.325,148.684
C00712=1232.327,21.707,-42.221,-179.208,5.324,148.685
C00713=1232.333,21.458,-42.206,-179.210,5.324,148.685
C00714=1232.337,21.208,-42.190,-179.213,5.323,148.686
C00715=1232.342,20.958,-42.175,-179.215,5.323,148.687
C00716=1232.347,20.709,-42.160,-179.218,5.323,148.687
C00717=1232.352,20.460,-42.144,-179.220,5.322,148.688
C00718=1232.358,20.210,-42.129,-179.223,5.322,148.689
C00719=1232.362,19.960,-42.114,-179.225,5.322,148.689
C00720=1232.367,19.711,-42.098,-179.228,5.321,148.690
C00721=1232.372,19.462,-42.083,-179.230,5.321,148.691
C00722=1232.377,19.212,-42.068,-179.233,5.320,148.692
C00723=1232.382,18.963,-42.053,-179.236,5.320,148.692
C00724=1232.387,18.713,-42.037,-179.238,5.320,148.693
C00725=1232.392,18.464,-42.021,-179.240,5.319,148.694
C00726=1232.397,18.214,-42.007,-179.243,5.319,148.694
C00727=1232.402,17.964,-41.991,-179.246,5.318,148.695
C00728=1232.407,17.715,-41.976,-179.248,5.319,148.696
C00729=1232.412,17.466,-41.961,-179.250,5.318,148.696
C00730=1232.416,17.216,-41.945,-179.253,5.318,148.697
C00731=1232.422,16.966,-41.931,-179.256,5.317,148.698
C00732=1232.427,16.717,-41.916,-179.258,5.316,148.698
C00733=1232.432,16.468,-41.900,-179.260,5.317,148.699
C00734=1232.437,16.219,-41.885,-179.263,5.316,148.700
C00735=1232.442,15.969,-41.869,-179.266,5.316,148.700
C00736=1232.447,15.719,-41.855,-179.268,5.315,148.701
C00737=1232.452,15.469,-41.839,-179.270,5.315,148.702
C00738=1232.457,15.220,-41.824,-179.273,5.315,148.702
C00739=1232.462,14.971,-41.809,-179.276,5.314,148.703
C00740=1232.467,14.721,-41.794,-179.278,5.314,148.704
C00741=1232.472,14.472,-41.779,-179.280,5.314,148.705
C00742=1232.477,14.223,-41.764,-179.283,5.313,148.705
C00743=1232.482,13.973,-41.749,-179.286,5.313,148.706
C00744=1232.487,13.723,-41.734,-179.288,5.312,148.707
C00745=1232.491,13.474,-41.719,-179.290,5.313,148.707
C00746=1232.497,13.224,-41.703,-179.293,5.312,148.708
C00747=1232.502,12.975,-41.689,-179.296,5.312,148.709
C00748=1232.507,12.725,-41.673,-179.298,5.311,148.709
C00749=1232.512,12.476,-41.658,-179.300,5.311,148.710
C00750=1232.517,12.226,-41.644,-179.303,5.311,148.711
C00751=1232.522,11.977,-41.628,-179.306,5.310,148.711
C00752=1232.527,11.728,-41.613,-179.308,5.310,148.712
C00753=1232.532,11.478,-41.598,-179.310,5.310,148.713
C00754=1232.536,11.228,-41.583,-179.313,5.309,148.713
C00755=1232.541,10.978,-41.569,-179.316,5.309,148.714
C00756=1232.547,10.729,-41.553,-179.318,5.308,148.715
C00757=1232.551,10.480,-41.538,-179.320,5.309,148.715
C00758=1232.556,10.230,-41.524,-179.323,5.308,148.716
C00759=1232.562,9.981,-41.508,-179.326,5.307,148.717
C00760=1232.567,9.731,-41.494,-179.328,5.307,148.718
C00761=1232.571,9.482,-41.479,-179.330,5.307,148.718
C00762=1232.577,9.232,-41.464,-179.333,5.307,148.719
C00763=1232.582,8.983,-41.449,-179.336,5.306,148.720
C00764=1232.586,8.734,-41.434,-179.338,5.306,148.720
C00765=1232.592,8.484,-41.419,-179.341,5.306,148.721
C00766=1232.597,8.235,-41.404,-179.343,5.305,148.722
C00767=1232.602,7.985,-41.390,-179.346,5.305,148.722
C00768=1232.607,7.736,-41.374,-179.348,5.305,148.723
C00769=1232.612,7.486,-41.360,-179.351,5.305,148.724
C00770=1232.617,7.237,-41.345,-179.353,5.304,148.724
C00771=1232.622,6.987,-41.330,-179.356,5.303,148.725
C00772=1232.627,6.738,-41.315,-179.358,5.304,148.726
C00773=1232.632,6.488,-41.301,-179.361,5.303,148.726
C00774=1232.637,6.239,-41.286,-179.363,5.303,148.727
C00775=1232.642,5.989,-41.271,-179.366,5.302,148.728
C00776=1232.647,5.739,-41.257,-179.368,5.302,148.729
C00777=1232.652,5.490,-41.242,-179.371,5.302,148.729
C00778=1232.657,5.240,-41.228,-179.374,5.302,148.730
C00779=1232.662,4.991,-41.212,-179.376,5.301,148.731
C00780=1232.667,4.741,-41.198,-179.378,5.301,148.732
C00781=1232.672,4.492,-41.183,-179.381,5.301,148.732
C00782=1232.677,4.242,-41.168,-179.384,5.300,148.733
C00783=1232.683,3.973,-41.152,-179.386,5.300,148.734
C00784=1232.688,3.704,-41.136,-179.389,5.300,148.734
C00785=1232.693,3.436,-41.121,-179.391,5.300,148.735
C00786=1232.699,3.167,-41.104,-179.394,5.299,148.736
C00787=1232.704,2.917,-41.090,-179.397,5.299,148.737
C00788=1232.709,2.667,-41.076,-179.400,5.298,148.737
C00789=1232.713,2.418,-41.061,-179.402,5.299,148.738
C00790=1232.718,2.168,-41.047,-179.404,5.298,148.739
C00791=1232.724,1.918,-41.032,-179.407,5.298,148.739
C00792=1232.729,1.669,-41.017,-179.409,5.298,148.740
C00793=1232.734,1.420,-41.002,-179.412,5.297,148.741
C00794=1232.739,1.170,-40.988,-179.414,5.297,148.741
C00795=1232.744,0.921,-40.974,-179.416,5.297,148.742
C00796=1232.749,0.672,-40.959,-179.419,5.297,148.743
C00797=1232.754,0.422,-40.944,-179.422,5.296,148.743
C00798=1232.759,0.173,-40.929,-179.424,5.296,148.744
C00799=1232.764,-0.077,-40.915,-179.426,5.296,148.745
C00800=1232.769,-0.327,-40.901,-179.429,5.295,148.746
C00801=1232.774,-0.577,-40.887,-179.432,5.295,148.746
C00802=1232.779,-0.826,-40.872,-179.434,5.295,148.747
C00803=1232.784,-1.075,-40.857,-179.437,5.295,148.748
C00804=1232.788,-1.325,-40.843,-179.439,5.294,148.748
C00805=1232.794,-1.575,-40.828,-179.442,5.293,148.749
C00806=1232.800,-1.824,-40.814,-179.444,5.294,148.750
C00807=1232.804,-2.073,-40.799,-179.447,5.293,148.750
C00808=1232.809,-2.323,-40.785,-179.449,5.293,148.751
C00809=1232.814,-2.573,-40.771,-179.451,5.293,148.752
C00810=1232.819,-2.822,-40.756,-179.454,5.292,148.752
C00811=1232.824,-3.072,-40.742,-179.457,5.292,148.753
C00812=1232.829,-3.321,-40.727,-179.459,5.292,148.754
C00813=1232.834,-3.571,-40.713,-179.461,5.292,148.754
C00814=1232.839,-3.820,-40.699,-179.464,5.291,148.755
C00815=1232.844,-4.070,-40.685,-179.467,5.291,148.756
C00816=1232.849,-4.319,-40.670,-179.469,5.291,148.757
C00817=1232.854,-4.569,-40.656,-179.471,5.290,148.757
C00818=1232.859,-4.819,-40.642,-179.474,5.290,148.758
C00819=1232.864,-5.068,-40.627,-179.477,5.291,148.759
C00820=1232.869,-5.317,-40.613,-179.479,5.290,148.760
C00821=1232.874,-5.566,-40.599,-179.482,5.289,148.760
C00822=1232.879,-5.816,-40.584,-179.484,5.290,148.761
C00823=1232.884,-6.066,-40.570,-179.487,5.289,148.762
C00824=1232.889,-6.316,-40.556,-179.489,5.289,148.762
C00825=1232.894,-6.565,-40.542,-179.491,5.289,148.763
C00826=1232.899,-6.815,-40.527,-179.494,5.288,148.764
C00827=1232.905,-7.064,-40.513,-179.497,5.288,148.764
C00828=1232.910,-7.314,-40.499,-179.499,5.288,148.765
C00829=1232.915,-7.563,-40.485,-179.501,5.288,148.766
C00830=1232.920,-7.813,-40.471,-179.504,5.287,148.766
C00831=1232.924,-8.063,-40.456,-179.506,5.287,148.767
C00832=1232.930,-8.312,-40.442,-179.509,5.287,148.768
C00833=1232.935,-8.562,-40.428,-179.511,5.286,148.769
C00834=1232.940,-8.811,-40.414,-179.514,5.286,148.769
C00835=1232.945,-9.061,-40.400,-179.516,5.286,148.770
C00836=1232.950,-9.311,-40.385,-179.519,5.286,148.771
C00837=1232.955,-9.560,-40.371,-179.522,5.285,148.771
C00838=1232.960,-9.809,-40.357,-179.524,5.285,148.772
C00839=1232.965,-10.059,-40.343,-179.526,5.285,148.773
C00840=1232.970,-10.309,-40.329,-179.529,5.284,148.773
C00841=1232.975,-10.559,-40.314,-179.531,5.285,148.774
C00842=1232.981,-10.808,-40.300,-179.534,5.284,148.775
C00843=1232.985,-11.057,-40.287,-179.536,5.284,148.775
C00844=1232.990,-11.307,-40.272,-179.538,5.284,148.776
C00845=1232.995,-11.556,-40.258,-179.541,5.283,148.777
C00846=1233.000,-11.805,-40.244,-179.544,5.283,148.778
C00847=1233.005,-12.055,-40.230,-179.546,5.284,148.778
C00848=1233.010,-12.305,-40.216,-179.549,5.283,148.779
C00849=1233.015,-12.555,-40.201,-179.552,5.283,148.780
C00850=1233.021,-12.804,-40.188,-179.554,5.283,148.781
C00851=1233.025,-13.054,-40.174,-179.556,5.282,148.781
C00852=1233.030,-13.303,-40.160,-179.559,5.282,148.782
C00853=1233.036,-13.552,-40.146,-179.561,5.282,148.783
C00854=1233.041,-13.802,-40.132,-179.564,5.282,148.783
C00855=1233.046,-14.052,-40.118,-179.566,5.281,148.784
C00856=1233.051,-14.301,-40.103,-179.568,5.281,148.785
C00857=1233.056,-14.551,-40.091,-179.571,5.281,148.785
C00858=1233.061,-14.800,-40.077,-179.574,5.280,148.786
C00859=1233.066,-15.050,-40.062,-179.576,5.281,148.787
C00860=1233.071,-15.299,-40.048,-179.579,5.280,148.787
C00861=1233.076,-15.549,-40.034,-179.581,5.280,148.788
C00862=1233.081,-15.799,-40.021,-179.583,5.280,148.789
C00863=1233.086,-16.049,-40.007,-179.586,5.279,148.790
C00864=1233.091,-16.298,-39.993,-179.588,5.280,148.790
C00865=1233.096,-16.547,-39.979,-179.591,5.279,148.791
C00866=1233.101,-16.797,-39.964,-179.593,5.279,148.792
C00867=1233.106,-17.046,-39.952,-179.595,5.279,148.792
C00868=1233.111,-17.296,-39.938,-179.599,5.279,148.793
C00869=1233.116,-17.546,-39.923,-179.601,5.278,148.794
C00870=1233.122,-17.795,-39.910,-179.603,5.279,148.795
C00871=1233.126,-18.045,-39.896,-179.606,5.278,148.795
C00872=1233.131,-18.295,-39.882,-179.609,5.277,148.796
C00873=1233.137,-18.544,-39.868,-179.611,5.278,148.797
C00874=1233.142,-18.794,-39.855,-179.613,5.277,148.797
C00875=1233.147,-19.043,-39.841,-179.616,5.277,148.798
C00876=1233.152,-19.292,-39.827,-179.618,5.277,148.799
C00877=1233.157,-19.543,-39.813,-179.621,5.277,148.800
C00878=1233.163,-19.792,-39.800,-179.623,5.276,148.800
C00879=1233.167,-20.041,-39.786,-179.625,5.276,148.801
C00880=1233.172,-20.291,-39.772,-179.628,5.276,148.802
C00881=1233.178,-20.540,-39.758,-179.630,5.276,148.802
C00882=1233.182,-20.790,-39.745,-179.633,5.276,148.803
C00883=1233.187,-21.040,-39.731,-179.636,5.275,148.804
C00884=1233.193,-21.289,-39.717,-179.638,5.275,148.804
C00885=1233.197,-21.538,-39.704,-179.640,5.275,148.805
C00886=1233.203,-21.788,-39.690,-179.643,5.274,148.806
C00887=1233.208,-22.058,-39.675,-179.646,5.275,148.807
C00888=1233.214,-22.327,-39.660,-179.648,5.275,148.807
C00889=1233.219,-22.596,-39.645,-179.651,5.274,148.808
C00890=1233.225,-22.865,-39.631,-179.654,5.274,148.809
C00891=1233.230,-23.115,-39.618,-179.656,5.274,148.810
C00892=1233.235,-23.365,-39.604,-179.659,5.274,148.810
C00893=1233.240,-23.614,-39.591,-179.661,5.273,148.811
C00894=1233.245,-23.864,-39.577,-179.663,5.273,148.812
C00895=1233.250,-24.113,-39.564,-179.666,5.273,148.812
C00896=1233.255,-24.363,-39.550,-179.668,5.273,148.813
C00897=1233.260,-24.612,-39.536,-179.671,5.273,148.814
C00898=1233.265,-24.862,-39.523,-179.674,5.272,148.815
C00899=1233.270,-25.112,-39.509,-179.676,5.273,148.815
C00900=1233.275,-25.361,-39.496,-179.678,5.272,148.816
C00901=1233.280,-25.611,-39.482,-179.681,5.272,148.817
C00902=1233.286,-25.860,-39.469,-179.683,5.272,148.817
C00903=1233.290,-26.110,-39.455,-179.686,5.271,148.818
C00904=1233.296,-26.359,-39.442,-179.688,5.272,148.819
C00905=1233.300,-26.609,-39.429,-179.690,5.271,148.819
C00906=1233.306,-26.858,-39.415,-179.693,5.271,148.820
C00907=1233.311,-27.108,-39.402,-179.695,5.271,148.821
C00908=1233.315,-27.358,-39.388,-179.698,5.271,148.822
C00909=1233.321,-27.607,-39.375,-179.701,5.270,148.822
C00910=1233.326,-27.857,-39.361,-179.703,5.271,148.823
C00911=1233.331,-28.107,-39.347,-179.706,5.270,148.824
C00912=1233.336,-28.356,-39.334,-179.708,5.270,148.825
C00913=1233.342,-28.606,-39.321,-179.710,5.270,148.825
C00914=1233.346,-28.856,-39.308,-179.713,5.269,148.826
C00915=1233.352,-29.105,-39.294,-179.715,5.270,148.827
C00916=1233.356,-29.355,-39.281,-179.718,5.269,148.827
C00917=1233.362,-29.604,-39.267,-179.720,5.269,148.828
C00918=1233.366,-29.854,-39.254,-179.723,5.269,148.829
C00919=1233.372,-30.103,-39.241,-179.725,5.268,148.829
C00920=1233.376,-30.353,-39.227,-179.727,5.269,148.830
C00921=1233.382,-30.602,-39.214,-179.730,5.268,148.831
C00922=1233.387,-30.852,-39.201,-179.733,5.268,148.832
C00923=1233.392,-31.101,-39.187,-179.735,5.268,148.832
C00924=1233.397,-31.352,-39.174,-179.737,5.268,148.833
C00925=1233.402,-31.601,-39.161,-179.740,5.268,148.834
C00926=1233.407,-31.851,-39.147,-179.743,5.268,148.835
C00927=1233.412,-32.100,-39.134,-179.745,5.267,148.835
C00928=1233.418,-32.349,-39.121,-179.747,5.268,148.836
C00929=1233.422,-32.600,-39.108,-179.750,5.267,148.837
C00930=1233.428,-32.849,-39.094,-179.752,5.267,148.837
C00931=1233.432,-33.099,-39.081,-179.755,5.267,148.838
C00932=1233.438,-33.348,-39.068,-179.757,5.266,148.839
C00933=1233.442,-33.598,-39.055,-179.760,5.267,148.839
C00934=1233.448,-33.847,-39.042,-179.762,5.266,148.840
C00935=1233.453,-34.097,-39.028,-179.764,5.266,148.841
C00936=1233.458,-34.347,-39.016,-179.767,5.266,148.842
C00937=1233.464,-34.596,-39.002,-179.770,5.265,148.842
C00938=1233.468,-34.846,-38.989,-179.772,5.266,148.843
C00939=1233.473,-35.095,-38.976,-179.774,5.265,148.844
C00940=1233.478,-35.345,-38.963,-179.776,5.266,148.844
C00941=1233.484,-35.595,-38.950,-179.779,5.265,148.845
C00942=1233.489,-35.844,-38.936,-179.782,5.265,148.846
C00943=1233.494,-36.094,-38.923,-179.784,5.265,148.846
C00944=1233.499,-36.343,-38.911,-179.787,5.265,148.847
C00945=1233.504,-36.593,-38.897,-179.789,5.265,148.848
C00946=1233.509,-36.843,-38.885,-179.792,5.265,148.849
C00947=1233.514,-37.093,-38.872,-179.794,5.264,148.849
C00948=1233.519,-37.342,-38.858,-179.797,5.264,148.850
C00949=1233.524,-37.591,-38.845,-179.799,5.264,148.851
C00950=1233.529,-37.841,-38.832,-179.801,5.264,148.852
C00951=1233.535,-38.091,-38.819,-179.804,5.264,148.852
C00952=1233.540,-38.340,-38.806,-179.807,5.263,148.853
C00953=1233.544,-38.590,-38.793,-179.809,5.264,148.854
C00954=1233.550,-38.839,-38.780,-179.811,5.263,148.854
C00955=1233.555,-39.089,-38.767,-179.813,5.263,148.855
C00956=1233.560,-39.339,-38.755,-179.816,5.263,148.856
C00957=1233.565,-39.588,-38.741,-179.818,5.263,148.856
C00958=1233.570,-39.838,-38.728,-179.821,5.263,148.857
C00959=1233.575,-40.087,-38.715,-179.824,5.262,148.858
C00960=1233.580,-40.336,-38.702,-179.826,5.262,148.859
C00961=1233.585,-40.587,-38.689,-179.828,5.262,148.859
C00962=1233.591,-40.836,-38.676,-179.831,5.263,148.860
C00963=1233.596,-41.085,-38.664,-179.834,5.262,148.861
C00964=1233.600,-41.335,-38.651,-179.836,5.262,148.862
C00965=1233.606,-41.585,-38.638,-179.838,5.262,148.862
C00966=1233.611,-41.834,-38.625,-179.841,5.261,148.863
C00967=1233.616,-42.084,-38.612,-179.843,5.262,148.864
C00968=1233.621,-42.334,-38.599,-179.846,5.261,148.864
C00969=1233.627,-42.583,-38.586,-179.848,5.262,148.865
C00970=1233.631,-42.833,-38.573,-179.850,5.261,148.866
C00971=1233.636,-43.083,-38.561,-179.853,5.261,148.867
C00972=1233.642,-43.332,-38.548,-179.855,5.261,148.867
C00973=1233.647,-43.582,-38.534,-179.858,5.260,148.868
C00974=1233.652,-43.832,-38.522,-179.860,5.261,148.869
C00975=1233.657,-44.081,-38.509,-179.863,5.260,148.869
C00976=1233.662,-44.331,-38.496,-179.865,5.260,148.870
C00977=1233.667,-44.580,-38.484,-179.867,5.260,148.871
C00978=1233.673,-44.830,-38.470,-179.870,5.260,148.871
C00979=1233.678,-45.079,-38.458,-179.872,5.260,148.872
C00980=1233.682,-45.329,-38.445,-179.875,5.260,148.873
C00981=1233.688,-45.579,-38.433,-179.877,5.260,148.874
C00982=1233.693,-45.829,-38.420,-179.880,5.260,148.874
C00983=1233.697,-46.079,-38.407,-179.883,5.259,148.875
C00984=1233.703,-46.328,-38.394,-179.885,5.259,148.876
C00985=1233.708,-46.578,-38.382,-179.887,5.259,148.877
C00986=1233.713,-46.827,-38.369,-179.889,5.259,148.877
C00987=1233.718,-47.077,-38.356,-179.892,5.259,148.878
C00988=1233.723,-47.326,-38.343,-179.894,5.259,148.879
C00989=1233.728,-47.576,-38.332,-179.897,5.259,148.879
C00990=1233.734,-47.825,-38.319,-179.899,5.259,148.880
C00991=1233.739,-48.095,-38.305,-179.902,5.258,148.881
C00992=1233.744,-48.365,-38.291,-179.905,5.258,148.882
C00993=1233.751,-48.635,-38.277,-179.907,5.258,148.882
C00994=1233.756,-48.904,-38.263,-179.910,5.258,148.883
C00995=1233.761,-49.154,-38.252,-179.912,5.258,148.884
C00996=1233.766,-49.403,-38.239,-179.914,5.258,148.885
C00997=1233.771,-49.654,-38.226,-179.917,5.258,148.885
C00998=1233.776,-49.903,-38.213,-179.919,5.258,148.886
C00999=1233.781,-50.152,-38.201,-179.922,5.258,148.887
C01000=1233.786,-50.402,-38.189,-179.925,5.257,148.888
C01001=1233.791,-50.652,-38.176,-179.927,5.258,148.888
C01002=1233.796,-50.901,-38.163,-179.930,5.257,148.889
C01003=1233.802,-51.151,-38.150,-179.932,5.257,148.890
C01004=1233.807,-51.401,-38.138,-179.934,5.257,148.890
C01005=1233.812,-51.650,-38.126,-179.937,5.257,148.891
C01006=1233.817,-51.900,-38.113,-179.939,5.257,148.892
C01007=1233.822,-52.150,-38.101,-179.942,5.256,148.893
C01008=1233.828,-52.400,-38.088,-179.944,5.257,148.893
C01009=1233.833,-52.649,-38.076,-179.947,5.256,148.894
C01010=1233.838,-52.898,-38.063,-179.949,5.256,148.895
C01011=1233.843,-53.149,-38.051,-179.951,5.256,148.895
C01012=1233.848,-53.398,-38.038,-179.953,5.256,148.896
C01013=1233.853,-53.647,-38.026,-179.956,5.256,148.897
C01014=1233.858,-53.897,-38.014,-179.958,5.256,148.897
C01015=1233.863,-54.147,-38.001,-179.961,5.256,148.898
C01016=1233.869,-54.396,-37.988,-179.963,5.256,148.899
C01017=1233.873,-54.647,-37.976,-179.966,5.255,148.900
C01018=1233.878,-54.896,-37.964,-179.969,5.255,148.900
C01019=1233.884,-55.145,-37.951,-179.971,5.256,148.901
C01020=1233.889,-55.395,-37.939,-179.974,5.255,148.902
C01021=1233.893,-55.644,-37.927,-179.976,5.256,148.903
C01022=1233.899,-55.894,-37.915,-179.978,5.255,148.903
C01023=1233.904,-56.144,-37.903,-179.980,5.255,148.904
C01024=1233.909,-56.394,-37.890,-179.983,5.255,148.905
C01025=1233.914,-56.643,-37.878,-179.985,5.255,148.905
C01026=1233.919,-56.893,-37.865,-179.988,5.255,148.906
C01027=1233.924,-57.143,-37.853,-179.990,5.254,148.907
C01028=1233.930,-57.392,-37.841,-179.993,5.255,148.908
C01029=1233.935,-57.641,-37.828,-179.995,5.254,148.908
C01030=1233.940,-57.891,-37.816,-179.997,5.254,148.909
C01031=1233.945,-58.141,-37.804,-180.000,5.254,148.910
C01032=1233.950,-58.391,-37.791,179.998,5.254,148.910
C01033=1233.955,-58.641,-37.779,179.995,5.254,148.911
C01034=1233.960,-58.890,-37.767,179.993,5.254,148.912
C01035=1233.965,-59.140,-37.755,179.991,5.254,148.912
C01036=1233.970,-59.389,-37.743,179.988,5.254,148.913
C01037=1233.976,-59.639,-37.730,179.986,5.253,148.914
C01038=1233.981,-59.889,-37.718,179.983,5.254,148.915
C01039=1233.986,-60.138,-37.706,179.981,5.254,148.916
C01040=1233.992,-60.388,-37.694,179.978,5.253,148.916
C01041=1233.997,-60.637,-37.681,179.976,5.254,148.917
C01042=1234.001,-60.887,-37.670,179.973,5.253,148.918
C01043=1234.006,-61.137,-37.657,179.971,5.253,148.918
C01044=1234.011,-61.387,-37.645,179.968,5.253,148.919
C01045=1234.016,-61.636,-37.633,179.966,5.253,148.920
C01046=1234.022,-61.886,-37.621,179.964,5.253,148.920
C01047=1234.027,-62.136,-37.609,179.961,5.253,148.921
C01048=1234.032,-62.385,-37.597,179.959,5.253,148.922
C01049=1234.037,-62.635,-37.585,179.957,5.253,148.923
C01050=1234.042,-62.884,-37.572,179.954,5.252,148.923
C01051=1234.048,-63.134,-37.561,179.952,5.253,148.924
C01052=1234.053,-63.384,-37.548,179.949,5.252,148.925
C01053=1234.058,-63.633,-37.537,179.947,5.253,148.925
C01054=1234.063,-63.883,-37.525,179.945,5.252,148.926
C01055=1234.068,-64.132,-37.512,179.942,5.252,148.927
C01056=1234.074,-64.382,-37.500,179.940,5.252,148.928
C01057=1234.079,-64.632,-37.488,179.937,5.252,148.928
C01058=1234.083,-64.881,-37.476,179.935,5.252,148.929
C01059=1234.089,-65.131,-37.464,179.932,5.251,148.930
C01060=1234.094,-65.381,-37.452,179.930,5.252,148.930
C01061=1234.099,-65.631,-37.440,179.927,5.252,148.931
C01062=1234.104,-65.880,-37.429,179.925,5.252,148.932
C01063=1234.109,-66.130,-37.417,179.922,5.252,148.933
C01064=1234.115,-66.379,-37.404,179.920,5.252,148.933
C01065=1234.120,-66.629,-37.392,179.918,5.251,148.934
C01066=1234.125,-66.879,-37.381,179.916,5.252,148.935
C01067=1234.130,-67.128,-37.368,179.913,5.251,148.936
C01068=1234.135,-67.378,-37.357,179.911,5.252,148.936
C01069=1234.141,-67.628,-37.345,179.908,5.251,148.937
C01070=1234.145,-67.877,-37.333,179.906,5.251,148.938
C01071=1234.150,-68.127,-37.321,179.903,5.251,148.938
C01072=1234.156,-68.377,-37.309,179.901,5.251,148.939
C01073=1234.161,-68.627,-37.298,179.899,5.251,148.940
C01074=1234.166,-68.876,-37.285,179.896,5.251,148.940
C01075=1234.171,-69.126,-37.273,179.894,5.251,148.941
C01076=1234.176,-69.376,-37.262,179.891,5.250,148.942
C01077=1234.181,-69.625,-37.250,179.889,5.251,148.943
C01078=1234.187,-69.875,-37.238,179.886,5.250,148.943
C01079=1234.191,-70.124,-37.226,179.884,5.250,148.944
C01080=1234.197,-70.374,-37.214,179.882,5.250,148.945
C01081=1234.202,-70.624,-37.202,179.880,5.250,148.945
C01082=1234.207,-70.874,-37.191,179.877,5.250,148.946
C01083=1234.213,-71.123,-37.179,179.875,5.250,148.947
C01084=1234.218,-71.372,-37.167,179.872,5.250,148.948
C01085=1234.222,-71.622,-37.156,179.870,5.250,148.948
C01086=1234.228,-71.872,-37.144,179.867,5.250,148.949
C01087=1234.233,-72.122,-37.132,179.865,5.250,148.950
C01088=1234.238,-72.372,-37.121,179.862,5.250,148.951
C01089=1234.243,-72.622,-37.109,179.860,5.250,148.951
C01090=1234.249,-72.871,-37.097,179.857,5.250,148.952
C01091=1234.253,-73.120,-37.085,179.855,5.250,148.953
C01092=1234.259,-73.370,-37.073,179.853,5.250,148.953
C01093=1234.263,-73.620,-37.062,179.850,5.250,148.954
C01094=1234.269,-73.869,-37.050,179.848,5.249,148.955
C01095=1234.275,-74.140,-37.037,179.846,5.250,148.956
C01096=1234.280,-74.411,-37.025,179.843,5.249,148.956
C01097=1234.286,-74.680,-37.012,179.840,5.249,148.957
C01098=1234.292,-74.951,-36.999,179.838,5.250,148.958
C01099=1234.296,-75.200,-36.988,179.835,5.249,148.959
C01100=1234.302,-75.450,-36.976,179.833,5.249,148.959
C01101=1234.307,-75.700,-36.964,179.830,5.249,148.960
C01102=1234.312,-75.949,-36.953,179.828,5.249,148.961
C01103=1234.318,-76.199,-36.941,179.826,5.249,148.961
C01104=1234.323,-76.449,-36.930,179.823,5.249,148.962
C01105=1234.328,-76.699,-36.918,179.821,5.249,148.963
C01106=1234.333,-76.948,-36.907,179.819,5.249,148.964
C01107=1234.338,-77.198,-36.895,179.816,5.249,148.964
C01108=1234.343,-77.448,-36.884,179.814,5.249,148.965
C01109=1234.349,-77.697,-36.872,179.811,5.248,148.966
C01110=1234.353,-77.947,-36.861,179.809,5.249,148.966
C01111=1234.359,-78.197,-36.849,179.807,5.248,148.967
C01112=1234.364,-78.446,-36.838,179.804,5.249,148.968
C01113=1234.369,-78.696,-36.826,179.802,5.248,148.969
C01114=1234.374,-78.946,-36.815,179.800,5.249,148.969
C01115=1234.380,-79.195,-36.803,179.797,5.248,148.970
C01116=1234.384,-79.445,-36.792,179.795,5.248,148.971
C01117=1234.390,-79.695,-36.780,179.792,5.248,148.971
C01118=1234.395,-79.944,-36.769,179.790,5.248,148.972
C01119=1234.400,-80.194,-36.757,179.787,5.248,148.973
C01120=1234.405,-80.444,-36.745,179.785,5.248,148.974
C01121=1234.411,-80.693,-36.734,179.783,5.248,148.974
C01122=1234.416,-80.943,-36.723,179.781,5.248,148.975
C01123=1234.421,-81.193,-36.711,179.778,5.248,148.976
C01124=1234.426,-81.443,-36.700,179.776,5.248,148.976
C01125=1234.431,-81.692,-36.689,179.773,5.247,148.977
C01126=1234.437,-81.942,-36.677,179.771,5.248,148.978
C01127=1234.441,-82.191,-36.666,179.768,5.247,148.979
C01128=1234.447,-82.441,-36.654,179.766,5.248,148.979
C01129=1234.451,-82.691,-36.643,179.764,5.247,148.980
C01130=1234.458,-82.941,-36.632,179.762,5.248,148.981
C01131=1234.462,-83.190,-36.621,179.759,5.247,148.981
C01132=1234.467,-83.440,-36.610,179.757,5.247,148.982
C01133=1234.473,-83.690,-36.598,179.754,5.247,148.983
C01134=1234.477,-83.939,-36.586,179.752,5.248,148.984
C01135=1234.483,-84.188,-36.575,179.749,5.247,148.984
C01136=1234.488,-84.439,-36.564,179.747,5.248,148.985
C01137=1234.493,-84.689,-36.553,179.744,5.247,148.986
C01138=1234.498,-84.939,-36.541,179.742,5.248,148.987
C01139=1234.504,-85.187,-36.530,179.739,5.247,148.987
C01140=1234.508,-85.437,-36.519,179.737,5.247,148.988
C01141=1234.514,-85.688,-36.508,179.735,5.247,148.989
C01142=1234.519,-85.937,-36.496,179.732,5.247,148.989
C01143=1234.524,-86.186,-36.485,179.730,5.247,148.990
C01144=1234.530,-86.436,-36.474,179.728,5.247,148.991
C01145=1234.535,-86.686,-36.463,179.725,5.247,148.992
C01146=1234.539,-86.936,-36.452,179.723,5.247,148.992
C01147=1234.545,-87.185,-36.440,179.720,5.247,148.993
C01148=1234.550,-87.435,-36.429,179.718,5.247,148.994
C01149=1234.555,-87.685,-36.418,179.716,5.247,148.994
C01150=1234.561,-87.934,-36.407,179.713,5.247,148.995
C01151=1234.566,-88.184,-36.396,179.711,5.246,148.996
C01152=1234.571,-88.434,-36.385,179.709,5.247,148.996
C01153=1234.576,-88.683,-36.374,179.706,5.246,148.997
C01154=1234.581,-88.933,-36.362,179.704,5.247,148.998
C01155=1234.586,-89.183,-36.352,179.702,5.247,148.999
C01156=1234.591,-89.433,-36.340,179.699,5.247,148.999
C01157=1234.597,-89.682,-36.329,179.697,5.247,149.000
C01158=1234.602,-89.932,-36.318,179.694,5.246,149.001
C01159=1234.607,-90.182,-36.307,179.692,5.247,149.001
C01160=1234.612,-90.431,-36.296,179.690,5.246,149.002
C01161=1234.618,-90.681,-36.285,179.688,5.247,149.003
C01162=1234.622,-90.931,-36.274,179.685,5.246,149.004
C01163=1234.628,-91.180,-36.263,179.683,5.247,149.004
C01164=1234.633,-91.430,-36.252,179.680,5.246,149.005
C01165=1234.638,-91.680,-36.240,179.678,5.246,149.006
C01166=1234.644,-91.930,-36.230,179.675,5.246,149.006
C01167=1234.649,-92.179,-36.219,179.673,5.246,149.007
C01168=1234.653,-92.429,-36.207,179.671,5.246,149.008
C01169=1234.660,-92.679,-36.197,179.668,5.246,149.009
C01170=1234.664,-92.928,-36.185,179.666,5.246,149.009
C01171=1234.669,-93.179,-36.175,179.664,5.246,149.010
C01172=1234.675,-93.428,-36.164,179.661,5.246,149.011
C01173=1234.679,-93.677,-36.152,179.659,5.246,149.011
C01174=1234.686,-93.927,-36.142,179.656,5.246,149.012
C01175=1234.690,-94.177,-36.130,179.654,5.246,149.013
C01176=1234.695,-94.427,-36.120,179.651,5.246,149.014
C01177=1234.701,-94.676,-36.109,179.649,5.246,149.014
C01178=1234.706,-94.926,-36.098,179.647,5.245,149.015
C01179=1234.710,-95.176,-36.087,179.645,5.245,149.015
C01180=1234.717,-95.426,-36.076,179.643,5.246,149.016
C01181=1234.721,-95.675,-36.065,179.640,5.245,149.017
C01182=1234.727,-95.925,-36.055,179.638,5.246,149.018
C01183=1234.732,-96.174,-36.043,179.636,5.245,149.018
C01184=1234.737,-96.425,-36.033,179.633,5.246,149.019
C01185=1234.742,-96.674,-36.022,179.631,5.245,149.020
C01186=1234.747,-96.924,-36.011,179.629,5.245,149.020
C01187=1234.753,-97.173,-36.000,179.626,5.245,149.021
C01188=1234.758,-97.423,-35.989,179.624,5.245,149.022
C01189=1234.763,-97.673,-35.979,179.621,5.245,149.023
C01190=1234.768,-97.923,-35.968,179.619,5.245,149.023
C01191=1234.773,-98.173,-35.957,179.616,5.245,149.024
C01192=1234.778,-98.422,-35.946,179.614,5.245,149.025
C01193=1234.783,-98.672,-35.936,179.612,5.245,149.025
C01194=1234.789,-98.921,-35.925,179.610,5.245,149.026
C01195=1234.794,-99.171,-35.914,179.607,5.245,149.027
C01196=1234.800,-99.421,-35.903,179.605,5.245,149.028
C01197=1234.805,-99.671,-35.892,179.603,5.245,149.028
C01198=1234.810,-99.921,-35.882,179.600,5.245,149.029
C01199=1234.815,-100.191,-35.870,179.597,5.244,149.030
C01200=1234.821,-100.462,-35.859,179.595,5.245,149.031
C01201=1234.826,-100.733,-35.847,179.592,5.245,149.031
C01202=1234.832,-101.003,-35.835,179.590,5.245,149.032
C01203=1234.837,-101.254,-35.825,179.587,5.245,149.033
C01204=1234.843,-101.503,-35.814,179.585,5.245,149.034
C01205=1234.848,-101.753,-35.803,179.583,5.245,149.034
C01206=1234.853,-102.002,-35.793,179.580,5.245,149.035
C01207=1234.858,-102.253,-35.782,179.578,5.245,149.036
C01208=1234.863,-102.501,-35.771,179.576,5.245,149.036
C01209=1234.868,-102.752,-35.761,179.573,5.244,149.037
C01210=1234.874,-103.001,-35.751,179.571,5.245,149.038
C01211=1234.879,-103.252,-35.740,179.569,5.245,149.039
C01212=1234.884,-103.500,-35.729,179.566,5.245,149.039
C01213=1234.889,-103.751,-35.718,179.564,5.245,149.040
C01214=1234.895,-104.000,-35.708,179.561,5.245,149.041
C01215=1234.900,-104.250,-35.697,179.559,5.245,149.041
C01216=1234.905,-104.499,-35.687,179.557,5.245,149.042
C01217=1234.910,-104.750,-35.676,179.555,5.245,149.043
C01218=1234.916,-104.999,-35.666,179.552,5.244,149.043
C01219=1234.920,-105.249,-35.655,179.550,5.244,149.044
C01220=1234.926,-105.498,-35.645,179.548,5.244,149.045
C01221=1234.931,-105.749,-35.634,179.546,5.244,149.045
C01222=1234.937,-105.998,-35.624,179.543,5.244,149.046
C01223=1234.942,-106.248,-35.613,179.541,5.244,149.047
C01224=1234.947,-106.497,-35.602,179.539,5.245,149.048
C01225=1234.952,-106.748,-35.592,179.536,5.244,149.048
C01226=1234.958,-106.997,-35.581,179.534,5.245,149.049
C01227=1234.963,-107.247,-35.571,179.531,5.244,149.050
C01228=1234.968,-107.497,-35.561,179.529,5.244,149.050
C01229=1234.973,-107.747,-35.549,179.526,5.244,149.051
C01230=1234.978,-107.996,-35.540,179.524,5.244,149.052
C01231=1234.983,-108.245,-35.530,179.522,5.244,149.053
C01232=1234.988,-108.496,-35.519,179.520,5.244,149.053
C01233=1234.994,-108.745,-35.509,179.517,5.244,149.054
C01234=1234.999,-108.995,-35.498,179.515,5.244,149.055
C01235=1235.004,-109.245,-35.488,179.513,5.245,149.055
C01236=1235.009,-109.494,-35.477,179.510,5.244,149.056
C01237=1235.015,-109.744,-35.466,179.508,5.245,149.057
C01238=1235.020,-109.994,-35.456,179.505,5.244,149.058
C01239=1235.025,-110.244,-35.446,179.504,5.244,149.058
C01240=1235.030,-110.493,-35.436,179.501,5.244,149.059
C01241=1235.035,-110.743,-35.426,179.499,5.244,149.060
C01242=1235.041,-110.993,-35.415,179.496,5.244,149.060
C01243=1235.046,-111.243,-35.405,179.494,5.244,149.061
C01244=1235.051,-111.493,-35.395,179.491,5.243,149.062
C01245=1235.057,-111.742,-35.384,179.489,5.244,149.062
C01246=1235.061,-111.992,-35.374,179.487,5.244,149.063
C01247=1235.067,-112.241,-35.363,179.485,5.244,149.064
C01248=1235.072,-112.491,-35.353,179.482,5.244,149.065
C01249=1235.077,-112.741,-35.343,179.480,5.244,149.065
C01250=1235.083,-112.990,-35.332,179.478,5.244,149.066
C01251=1235.088,-113.241,-35.322,179.475,5.244,149.067
C01252=1235.093,-113.490,-35.312,179.473,5.244,149.067
C01253=1235.098,-113.739,-35.302,179.470,5.244,149.068
C01254=1235.103,-113.990,-35.291,179.468,5.244,149.069
C01255=1235.109,-114.239,-35.281,179.466,5.243,149.069
C01256=1235.114,-114.489,-35.271,179.464,5.243,149.070
C01257=1235.119,-114.739,-35.261,179.462,5.244,149.071
C01258=1235.124,-114.988,-35.251,179.459,5.243,149.071
C01259=1235.130,-115.238,-35.241,179.457,5.244,149.072
C01260=1235.135,-115.488,-35.230,179.454,5.243,149.073
C01261=1235.141,-115.738,-35.221,179.452,5.244,149.074
C01262=1235.146,-115.987,-35.211,179.450,5.243,149.074
C01263=1235.151,-116.238,-35.200,179.447,5.244,149.075
C01264=1235.156,-116.487,-35.190,179.445,5.243,149.076
C01265=1235.162,-116.737,-35.180,179.443,5.244,149.076
C01266=1235.166,-116.987,-35.170,179.441,5.244,149.077
C01267=1235.172,-117.236,-35.160,179.438,5.244,149.078
C01268=1235.177,-117.486,-35.150,179.436,5.244,149.078
C01269=1235.182,-117.736,-35.140,179.434,5.243,149.079
C01270=1235.187,-117.985,-35.129,179.432,5.243,149.080
C01271=1235.193,-118.235,-35.119,179.429,5.243,149.081
C01272=1235.198,-118.485,-35.109,179.427,5.243,149.081
C01273=1235.203,-118.735,-35.100,179.424,5.243,149.082
C01274=1235.209,-118.984,-35.089,179.422,5.243,149.083
C01275=1235.214,-119.235,-35.079,179.419,5.243,149.083
C01276=1235.218,-119.484,-35.069,179.417,5.243,149.084
C01277=1235.224,-119.733,-35.059,179.415,5.244,149.085
C01278=1235.229,-119.984,-35.049,179.412,5.243,149.086
C01279=1235.234,-120.233,-35.039,179.410,5.244,149.086
C01280=1235.240,-120.483,-35.029,179.408,5.243,149.087
C01281=1235.245,-120.733,-35.019,179.406,5.243,149.087
C01282=1235.250,-120.983,-35.009,179.403,5.243,149.088
C01283=1235.255,-121.232,-34.999,179.401,5.243,149.089
C01284=1235.261,-121.482,-34.989,179.399,5.243,149.090
C01285=1235.266,-121.731,-34.980,179.396,5.243,149.090
C01286=1235.271,-121.982,-34.969,179.394,5.243,149.091
C01287=1235.277,-122.231,-34.959,179.392,5.243,149.092
C01288=1235.281,-122.480,-34.950,179.390,5.243,149.092
C01289=1235.287,-122.730,-34.939,179.387,5.243,149.093
C01290=1235.292,-122.981,-34.929,179.385,5.243,149.094
C01291=1235.297,-123.230,-34.920,179.383,5.242,149.094
C01292=1235.303,-123.480,-34.910,179.381,5.243,149.095
C01293=1235.308,-123.729,-34.900,179.378,5.243,149.096
C01294=1235.313,-123.980,-34.890,179.376,5.243,149.097
C01295=1235.319,-124.229,-34.880,179.374,5.243,149.097
C01296=1235.323,-124.479,-34.870,179.371,5.243,149.098
C01297=1235.329,-124.728,-34.860,179.369,5.243,149.099
C01298=1235.334,-124.979,-34.851,179.366,5.243,149.099
C01299=1235.339,-125.228,-34.841,179.364,5.243,149.100
C01300=1235.345,-125.478,-34.830,179.362,5.242,149.101
C01301=1235.350,-125.728,-34.822,179.360,5.243,149.101
C01302=1235.356,-125.977,-34.811,179.358,5.243,149.102
C01303=1234.933,-125.988,-34.847,179.353,5.246,149.104
C01304=1234.928,-125.739,-34.856,179.355,5.246,149.103
C01305=1234.923,-125.488,-34.867,179.357,5.246,149.103
C01306=1234.918,-125.239,-34.876,179.360,5.246,149.102
C01307=1234.912,-124.989,-34.886,179.362,5.246,149.101
C01308=1234.907,-124.740,-34.896,179.365,5.246,149.101
C01309=1234.901,-124.490,-34.905,179.367,5.246,149.100
C01310=1234.896,-124.239,-34.916,179.369,5.247,149.099
C01311=1234.892,-123.990,-34.925,179.371,5.246,149.099
C01312=1234.886,-123.741,-34.935,179.373,5.246,149.098
C01313=1234.880,-123.490,-34.945,179.376,5.246,149.097
C01314=1234.876,-123.241,-34.955,179.378,5.246,149.097
C01315=1234.870,-122.991,-34.965,179.381,5.246,149.096
C01316=1234.865,-122.742,-34.975,179.383,5.246,149.095
C01317=1234.859,-122.492,-34.984,179.386,5.246,149.094
C01318=1234.854,-122.241,-34.995,179.387,5.246,149.094
C01319=1234.850,-121.992,-35.004,179.390,5.247,149.093
C01320=1234.844,-121.743,-35.015,179.392,5.247,149.092
C01321=1234.838,-121.492,-35.024,179.394,5.246,149.092
C01322=1234.834,-121.242,-35.034,179.397,5.247,149.091
C01323=1234.828,-120.993,-35.044,179.399,5.246,149.090
C01324=1234.823,-120.744,-35.054,179.402,5.247,149.090
C01325=1234.818,-120.493,-35.064,179.404,5.246,149.089
C01326=1234.813,-120.243,-35.074,179.406,5.247,149.088
C01327=1234.808,-119.994,-35.084,179.408,5.246,149.087
C01328=1234.802,-119.745,-35.094,179.411,5.247,149.087
C01329=1234.797,-119.494,-35.104,179.413,5.247,149.086
C01330=1234.791,-119.245,-35.115,179.415,5.246,149.086
C01331=1234.787,-118.996,-35.124,179.417,5.247,149.085
C01332=1234.782,-118.745,-35.135,179.420,5.246,149.084
C01333=1234.776,-118.495,-35.144,179.422,5.247,149.083
C01334=1234.771,-118.246,-35.154,179.424,5.247,149.083
C01335=1234.765,-117.996,-35.164,179.427,5.247,149.082
C01336=1234.760,-117.746,-35.175,179.429,5.247,149.081
C01337=1234.755,-117.497,-35.184,179.432,5.247,149.080
C01338=1234.750,-117.247,-35.194,179.434,5.247,149.080
C01339=1234.745,-116.997,-35.205,179.436,5.246,149.079
C01340=1234.739,-116.748,-35.215,179.438,5.247,149.079
C01341=1234.734,-116.498,-35.225,179.440,5.247,149.078
C01342=1234.729,-116.248,-35.235,179.443,5.247,149.077
C01343=1234.723,-115.998,-35.245,179.445,5.247,149.076
C01344=1234.718,-115.748,-35.255,179.448,5.247,149.076
C01345=1234.714,-115.498,-35.265,179.450,5.247,149.075
C01346=1234.708,-115.249,-35.275,179.453,5.247,149.074
C01347=1234.702,-114.999,-35.286,179.455,5.247,149.074
C01348=1234.697,-114.749,-35.296,179.457,5.247,149.073
C01349=1234.692,-114.500,-35.306,179.459,5.247,149.072
C01350=1234.687,-114.250,-35.316,179.461,5.247,149.071
C01351=1234.682,-114.000,-35.326,179.464,5.247,149.071
C01352=1234.676,-113.751,-35.337,179.466,5.247,149.070
C01353=1234.671,-113.500,-35.347,179.469,5.247,149.069
C01354=1234.666,-113.251,-35.357,179.471,5.247,149.069
C01355=1234.661,-113.001,-35.367,179.473,5.248,149.068
C01356=1234.656,-112.751,-35.378,179.475,5.247,149.067
C01357=1234.650,-112.502,-35.388,179.478,5.248,149.067
C01358=1234.645,-112.252,-35.398,179.480,5.247,149.066
C01359=1234.640,-112.002,-35.409,179.482,5.247,149.065
C01360=1234.635,-111.753,-35.418,179.485,5.247,149.064
C01361=1234.630,-111.502,-35.429,179.487,5.247,149.064
C01362=1234.625,-111.254,-35.440,179.490,5.247,149.063
C01363=1234.619,-111.004,-35.450,179.492,5.247,149.062
C01364=1234.614,-110.754,-35.461,179.494,5.247,149.062
C01365=1234.608,-110.504,-35.471,179.496,5.247,149.061
C01366=1234.603,-110.254,-35.481,179.499,5.248,149.060
C01367=1234.598,-110.005,-35.491,179.501,5.247,149.059
C01368=1234.593,-109.755,-35.501,179.504,5.248,149.059
C01369=1234.588,-109.505,-35.512,179.506,5.248,149.058
C01370=1234.582,-109.255,-35.522,179.508,5.247,149.058
C01371=1234.577,-109.005,-35.533,179.510,5.248,149.057
C01372=1234.572,-108.756,-35.543,179.512,5.247,149.056
C01373=1234.567,-108.506,-35.554,179.515,5.248,149.055
C01374=1234.561,-108.256,-35.564,179.517,5.247,149.055
C01375=1234.556,-108.007,-35.574,179.520,5.248,149.054
C01376=1234.552,-107.757,-35.584,179.522,5.248,149.053
C01377=1234.546,-107.507,-35.595,179.525,5.248,149.053
C01378=1234.541,-107.257,-35.605,179.527,5.248,149.052
C01379=1234.536,-107.008,-35.616,179.529,5.248,149.051
C01380=1234.531,-106.758,-35.627,179.531,5.248,149.050
C01381=1234.525,-106.508,-35.637,179.534,5.247,149.050
C01382=1234.520,-106.258,-35.647,179.536,5.248,149.049
C01383=1234.514,-106.009,-35.658,179.538,5.247,149.048
C01384=1234.510,-105.759,-35.669,179.541,5.248,149.048
C01385=1234.504,-105.509,-35.679,179.543,5.247,149.047
C01386=1234.499,-105.260,-35.689,179.546,5.248,149.046
C01387=1234.494,-105.010,-35.700,179.548,5.248,149.045
C01388=1234.488,-104.761,-35.711,179.551,5.248,149.045
C01389=1234.483,-104.511,-35.721,179.552,5.248,149.044
C01390=1234.478,-104.261,-35.732,179.555,5.248,149.044
C01391=1234.473,-104.011,-35.742,179.557,5.248,149.043
C01392=1234.467,-103.762,-35.753,179.560,5.249,149.042
C01393=1234.462,-103.512,-35.764,179.562,5.248,149.041
C01394=1234.457,-103.262,-35.774,179.564,5.248,149.041
C01395=1234.452,-103.012,-35.785,179.566,5.248,149.040
C01396=1234.446,-102.763,-35.795,179.569,5.248,149.039
C01397=1234.441,-102.513,-35.806,179.571,5.248,149.039
C01398=1234.436,-102.263,-35.816,179.573,5.248,149.038
C01399=1234.431,-102.013,-35.828,179.576,5.248,149.037
C01400=1234.426,-101.764,-35.838,179.578,5.248,149.036
C01401=1234.421,-101.514,-35.848,179.581,5.249,149.036
C01402=1234.416,-101.264,-35.860,179.583,5.248,149.035
C01403=1234.410,-101.014,-35.870,179.586,5.249,149.034
C01404=1234.405,-100.744,-35.881,179.588,5.248,149.034
C01405=1234.399,-100.473,-35.893,179.590,5.249,149.033
C01406=1234.393,-100.202,-35.905,179.593,5.248,149.032
C01407=1234.388,-99.931,-35.916,179.596,5.248,149.031
C01408=1234.383,-99.682,-35.927,179.598,5.249,149.030
C01409=1234.378,-99.431,-35.937,179.600,5.248,149.030
C01410=1234.372,-99.182,-35.948,179.602,5.248,149.029
C01411=1234.368,-98.932,-35.959,179.605,5.249,149.028
C01412=1234.362,-98.682,-35.970,179.607,5.248,149.028
C01413=1234.356,-98.433,-35.981,179.610,5.249,149.027
C01414=1234.351,-98.183,-35.991,179.612,5.248,149.026
C01415=1234.346,-97.934,-36.002,179.615,5.249,149.025
C01416=1234.341,-97.683,-36.013,179.617,5.248,149.025
C01417=1234.336,-97.434,-36.023,179.619,5.249,149.024
C01418=1234.331,-97.184,-36.034,179.622,5.248,149.023
C01419=1234.326,-96.934,-36.045,179.624,5.249,149.023
C01420=1234.321,-96.685,-36.056,179.626,5.249,149.022
C01421=1234.315,-96.435,-36.067,179.629,5.249,149.021
C01422=1234.310,-96.186,-36.078,179.631,5.249,149.020
C01423=1234.305,-95.935,-36.089,179.633,5.250,149.020
C01424=1234.300,-95.686,-36.100,179.635,5.249,149.019
C01425=1234.294,-95.436,-36.110,179.638,5.250,149.019
C01426=1234.290,-95.187,-36.121,179.640,5.249,149.018
C01427=1234.284,-94.937,-36.132,179.642,5.249,149.017
C01428=1234.279,-94.687,-36.144,179.645,5.249,149.016
C01429=1234.274,-94.437,-36.154,179.647,5.249,149.016
C01430=1234.268,-94.188,-36.165,179.650,5.249,149.015
C01431=1234.263,-93.938,-36.176,179.652,5.249,149.014
C01432=1234.258,-93.689,-36.187,179.654,5.250,149.014
C01433=1234.252,-93.438,-36.198,179.657,5.249,149.013
C01434=1234.248,-93.189,-36.209,179.659,5.250,149.012
C01435=1234.242,-92.939,-36.219,179.661,5.249,149.011
C01436=1234.237,-92.689,-36.231,179.664,5.250,149.011
C01437=1234.233,-92.440,-36.242,179.666,5.249,149.010
C01438=1234.226,-92.190,-36.253,179.669,5.250,149.009
C01439=1234.222,-91.940,-36.264,179.671,5.249,149.009
C01440=1234.217,-91.690,-36.274,179.673,5.250,149.008
C01441=1234.211,-91.441,-36.285,179.676,5.250,149.007
C01442=1234.206,-91.191,-36.297,179.678,5.250,149.006
C01443=1234.201,-90.941,-36.308,179.680,5.250,149.006
C01444=1234.196,-90.692,-36.319,179.683,5.250,149.005
C01445=1234.191,-90.442,-36.329,179.685,5.250,149.004
C01446=1234.185,-90.192,-36.341,179.688,5.250,149.004
C01447=1234.180,-89.943,-36.352,179.690,5.250,149.003
C01448=1234.175,-89.693,-36.363,179.693,5.250,149.002
C01449=1234.170,-89.443,-36.374,179.695,5.250,149.001
C01450=1234.164,-89.194,-36.386,179.697,5.250,149.001
C01451=1234.159,-88.944,-36.396,179.699,5.250,149.000
C01452=1234.154,-88.694,-36.407,179.701,5.250,148.999
C01453=1234.149,-88.445,-36.418,179.704,5.250,148.999
C01454=1234.143,-88.194,-36.429,179.706,5.250,148.998
C01455=1234.139,-87.945,-36.441,179.709,5.250,148.997
C01456=1234.133,-87.696,-36.452,179.711,5.250,148.996
C01457=1234.128,-87.445,-36.463,179.714,5.250,148.996
C01458=1234.123,-87.196,-36.474,179.716,5.250,148.995
C01459=1234.118,-86.946,-36.485,179.718,5.251,148.994
C01460=1234.112,-86.697,-36.497,179.721,5.250,148.994
C01461=1234.107,-86.447,-36.508,179.723,5.251,148.993
C01462=1234.103,-86.197,-36.519,179.725,5.250,148.992
C01463=1234.097,-85.947,-36.531,179.728,5.251,148.992
C01464=1234.092,-85.698,-36.542,179.730,5.250,148.991
C01465=1234.087,-85.448,-36.552,179.733,5.251,148.990
C01466=1234.081,-85.198,-36.564,179.735,5.251,148.989
C01467=1234.077,-84.948,-36.575,179.738,5.251,148.989
C01468=1234.071,-84.699,-36.586,179.740,5.251,148.988
C01469=1234.066,-84.449,-36.598,179.742,5.251,148.987
C01470=1234.061,-84.199,-36.609,179.744,5.251,148.987
C01471=1234.056,-83.950,-36.620,179.747,5.251,148.986
C01472=1234.050,-83.700,-36.632,179.749,5.251,148.985
C01473=1234.046,-83.451,-36.643,179.752,5.251,148.984
C01474=1234.040,-83.201,-36.655,179.754,5.251,148.984
C01475=1234.035,-82.951,-36.666,179.757,5.251,148.983
C01476=1234.030,-82.702,-36.676,179.759,5.251,148.982
C01477=1234.024,-82.452,-36.688,179.761,5.252,148.982
C01478=1234.020,-82.202,-36.699,179.763,5.251,148.981
C01479=1234.014,-81.952,-36.711,179.766,5.252,148.980
C01480=1234.010,-81.702,-36.723,179.768,5.251,148.979
C01481=1234.004,-81.454,-36.734,179.771,5.252,148.979
C01482=1233.999,-81.204,-36.745,179.773,5.251,148.978
C01483=1233.994,-80.953,-36.756,179.776,5.252,148.977
C01484=1233.989,-80.703,-36.768,179.778,5.252,148.977
C01485=1233.984,-80.454,-36.779,179.780,5.252,148.976
C01486=1233.978,-80.205,-36.791,179.782,5.252,148.975
C01487=1233.973,-79.955,-36.802,179.785,5.252,148.974
C01488=1233.968,-79.705,-36.814,179.788,5.251,148.974
C01489=1233.963,-79.455,-36.825,179.790,5.252,148.973
C01490=1233.958,-79.205,-36.837,179.793,5.252,148.972
C01491=1233.952,-78.957,-36.848,179.795,5.252,148.971
C01492=1233.947,-78.707,-36.860,179.797,5.252,148.971
C01493=1233.942,-78.457,-36.871,179.800,5.252,148.970
C01494=1233.937,-78.207,-36.883,179.802,5.252,148.969
C01495=1233.932,-77.957,-36.894,179.805,5.252,148.969
C01496=1233.927,-77.707,-36.906,179.807,5.252,148.968
C01497=1233.921,-77.459,-36.917,179.809,5.252,148.967
C01498=1233.916,-77.209,-36.929,179.812,5.252,148.966
C01499=1233.911,-76.959,-36.940,179.814,5.252,148.966
C01500=1233.906,-76.709,-36.952,179.816,5.252,148.965
C01501=1233.901,-76.459,-36.963,179.819,5.253,148.964
C01502=1233.896,-76.209,-36.975,179.821,5.252,148.964
C01503=1233.890,-75.961,-36.986,179.824,5.253,148.963
C01504=1233.885,-75.711,-36.998,179.826,5.252,148.962
C01505=1233.880,-75.461,-37.009,179.829,5.253,148.961
C01506=1233.875,-75.211,-37.021,179.831,5.252,148.961
C01507=1233.870,-74.961,-37.033,179.833,5.253,148.960
C01508=1233.865,-74.691,-37.046,179.835,5.253,148.959
C01509=1233.859,-74.421,-37.057,179.838,5.253,148.959
C01510=1233.853,-74.150,-37.070,179.841,5.253,148.958
C01511=1233.847,-73.881,-37.083,179.843,5.253,148.957
C01512=1233.842,-73.631,-37.095,179.846,5.253,148.956
C01513=1233.836,-73.381,-37.107,179.848,5.253,148.956
C01514=1233.832,-73.131,-37.118,179.851,5.253,148.955
C01515=1233.826,-72.881,-37.130,179.853,5.253,148.954
C01516=1233.822,-72.632,-37.141,179.856,5.254,148.953
C01517=1233.816,-72.382,-37.153,179.858,5.253,148.953
C01518=1233.811,-72.132,-37.166,179.860,5.254,148.952
C01519=1233.806,-71.883,-37.177,179.862,5.253,148.951
C01520=1233.801,-71.633,-37.189,179.865,5.254,148.951
C01521=1233.796,-71.383,-37.201,179.867,5.253,148.950
C01522=1233.790,-71.134,-37.212,179.870,5.254,148.949
C01523=1233.785,-70.884,-37.224,179.872,5.254,148.948
C01524=1233.780,-70.635,-37.236,179.875,5.254,148.948
C01525=1233.775,-70.385,-37.248,179.877,5.254,148.947
C01526=1233.770,-70.135,-37.259,179.879,5.254,148.946
C01527=1233.765,-69.886,-37.271,179.882,5.255,148.946
C01528=1233.759,-69.636,-37.283,179.884,5.254,148.945
C01529=1233.754,-69.386,-37.295,179.887,5.254,148.944
C01530=1233.750,-69.137,-37.306,179.889,5.254,148.943
C01531=1233.744,-68.887,-37.318,179.892,5.255,148.943
C01532=1233.739,-68.637,-37.330,179.894,5.254,148.942
C01533=1233.733,-68.387,-37.342,179.897,5.255,148.941
C01534=1233.729,-68.138,-37.354,179.899,5.254,148.940
C01535=1233.724,-67.888,-37.366,179.902,5.255,148.940
C01536=1233.718,-67.638,-37.378,179.904,5.255,148.939
C01537=1233.714,-67.389,-37.390,179.906,5.255,148.938
C01538=1233.708,-67.139,-37.402,179.908,5.255,148.938
C01539=1233.703,-66.889,-37.414,179.911,5.255,148.937
C01540=1233.697,-66.639,-37.426,179.913,5.255,148.936
C01541=1233.693,-66.390,-37.438,179.916,5.255,148.936
C01542=1233.688,-66.140,-37.449,179.918,5.255,148.935
C01543=1233.682,-65.890,-37.461,179.921,5.255,148.934
C01544=1233.677,-65.641,-37.474,179.923,5.255,148.933
C01545=1233.672,-65.391,-37.485,179.925,5.256,148.933
C01546=1233.667,-65.141,-37.497,179.927,5.255,148.932
C01547=1233.662,-64.892,-37.510,179.930,5.256,148.931
C01548=1233.656,-64.642,-37.522,179.933,5.256,148.931
C01549=1233.652,-64.393,-37.533,179.935,5.256,148.930
C01550=1233.647,-64.143,-37.546,179.937,5.256,148.929
C01551=1233.641,-63.893,-37.557,179.940,5.256,148.928
C01552=1233.636,-63.643,-37.569,179.942,5.256,148.928
C01553=1233.631,-63.394,-37.581,179.944,5.256,148.927
C01554=1233.626,-63.144,-37.593,179.947,5.257,148.926
C01555=1233.621,-62.895,-37.606,179.949,5.256,148.926
C01556=1233.615,-62.645,-37.618,179.952,5.256,148.925
C01557=1233.610,-62.395,-37.630,179.954,5.256,148.924
C01558=1233.605,-62.146,-37.642,179.957,5.257,148.923
C01559=1233.600,-61.896,-37.653,179.959,5.256,148.923
C01560=1233.595,-61.647,-37.666,179.962,5.257,148.922
C01561=1233.590,-61.397,-37.678,179.964,5.256,148.921
C01562=1233.584,-61.148,-37.691,179.967,5.257,148.920
C01563=1233.579,-60.898,-37.702,179.969,5.257,148.920
C01564=1233.574,-60.649,-37.715,179.971,5.257,148.919
C01565=1233.569,-60.399,-37.726,179.974,5.257,148.918
C01566=1233.564,-60.148,-37.739,179.976,5.257,148.918
C01567=1233.559,-59.899,-37.751,179.979,5.258,148.917
C01568=1233.554,-59.649,-37.763,179.981,5.257,148.916
C01569=1233.549,-59.400,-37.776,179.983,5.258,148.916
C01570=1233.543,-59.150,-37.788,179.986,5.257,148.915
C01571=1233.538,-58.900,-37.800,179.988,5.258,148.914
C01572=1233.533,-58.651,-37.811,179.990,5.258,148.913
C01573=1233.528,-58.401,-37.824,179.993,5.258,148.913
C01574=1233.523,-58.152,-37.837,179.995,5.258,148.912
C01575=1233.518,-57.902,-37.849,179.998,5.258,148.911
C01576=1233.513,-57.652,-37.861,-180.000,5.259,148.911
C01577=1233.508,-57.402,-37.873,-179.998,5.258,148.910
C01578=1233.503,-57.153,-37.886,-179.994,5.258,148.909
C01579=1233.497,-56.903,-37.898,-179.992,5.258,148.908
C01580=1233.492,-56.654,-37.910,-179.990,5.259,148.908
C01581=1233.487,-56.404,-37.923,-179.988,5.258,148.907
C01582=1233.482,-56.154,-37.935,-179.985,5.259,148.906
C01583=1233.476,-55.905,-37.948,-179.983,5.258,148.905
C01584=1233.472,-55.655,-37.959,-179.980,5.259,148.905
C01585=1233.467,-55.405,-37.972,-179.978,5.259,148.904
C01586=1233.462,-55.156,-37.984,-179.975,5.259,148.903
C01587=1233.457,-54.906,-37.996,-179.973,5.260,148.903
C01588=1233.452,-54.657,-38.009,-179.971,5.259,148.902
C01589=1233.446,-54.407,-38.021,-179.968,5.260,148.901
C01590=1233.441,-54.158,-38.033,-179.966,5.259,148.900
C01591=1233.436,-53.908,-38.046,-179.963,5.260,148.900
C01592=1233.431,-53.658,-38.058,-179.961,5.260,148.899
C01593=1233.426,-53.408,-38.071,-179.958,5.260,148.898
C01594=1233.421,-53.159,-38.083,-179.956,5.260,148.898
C01595=1233.415,-52.909,-38.095,-179.954,5.260,148.897
C01596=1233.411,-52.659,-38.108,-179.951,5.261,148.896
C01597=1233.406,-52.410,-38.121,-179.949,5.260,148.896
C01598=1233.401,-52.160,-38.133,-179.946,5.261,148.895
C01599=1233.395,-51.911,-38.145,-179.944,5.260,148.894
C01600=1233.390,-51.661,-38.158,-179.941,5.261,148.893
C01601=1233.385,-51.412,-38.171,-179.939,5.260,148.893
C01602=1233.380,-51.161,-38.183,-179.936,5.261,148.892
C01603=1233.375,-50.912,-38.195,-179.934,5.260,148.891
C01604=1233.370,-50.663,-38.208,-179.931,5.261,148.890
C01605=1233.364,-50.413,-38.221,-179.929,5.261,148.890
C01606=1233.359,-50.163,-38.233,-179.927,5.261,148.889
C01607=1233.354,-49.913,-38.246,-179.924,5.262,148.888
C01608=1233.349,-49.664,-38.259,-179.922,5.261,148.888
C01609=1233.344,-49.414,-38.271,-179.919,5.262,148.887
C01610=1233.339,-49.165,-38.284,-179.917,5.261,148.886
C01611=1233.334,-48.914,-38.296,-179.915,5.262,148.885
C01612=1233.328,-48.645,-38.309,-179.912,5.262,148.885
C01613=1233.322,-48.375,-38.324,-179.909,5.262,148.884
C01614=1233.317,-48.106,-38.337,-179.907,5.262,148.883
C01615=1233.312,-47.837,-38.351,-179.904,5.263,148.882
C01616=1233.306,-47.586,-38.364,-179.902,5.262,148.882
C01617=1233.301,-47.336,-38.376,-179.899,5.263,148.881
C01618=1233.296,-47.087,-38.389,-179.897,5.263,148.880
C01619=1233.291,-46.838,-38.401,-179.894,5.263,148.879
C01620=1233.286,-46.588,-38.414,-179.891,5.263,148.879
C01621=1233.281,-46.338,-38.427,-179.889,5.263,148.878
C01622=1233.276,-46.089,-38.440,-179.887,5.263,148.877
C01623=1233.270,-45.839,-38.453,-179.884,5.263,148.877
C01624=1233.265,-45.589,-38.465,-179.882,5.264,148.876
C01625=1233.260,-45.339,-38.478,-179.880,5.263,148.875
C01626=1233.255,-45.090,-38.490,-179.877,5.264,148.874
C01627=1233.250,-44.841,-38.503,-179.874,5.264,148.874
C01628=1233.246,-44.591,-38.516,-179.872,5.264,148.873
C01629=1233.240,-44.341,-38.529,-179.870,5.264,148.872
C01630=1233.235,-44.092,-38.542,-179.868,5.264,148.872
C01631=1233.230,-43.842,-38.554,-179.865,5.265,148.871
C01632=1233.225,-43.593,-38.567,-179.863,5.264,148.870
C01633=1233.220,-43.343,-38.580,-179.860,5.265,148.870
C01634=1233.215,-43.093,-38.593,-179.857,5.265,148.869
C01635=1233.209,-42.844,-38.606,-179.855,5.265,148.868
C01636=1233.204,-42.594,-38.618,-179.853,5.265,148.867
C01637=1233.199,-42.345,-38.631,-179.851,5.265,148.867
C01638=1233.195,-42.095,-38.644,-179.847,5.265,148.866
C01639=1233.189,-41.845,-38.657,-179.845,5.265,148.865
C01640=1233.184,-41.596,-38.670,-179.843,5.265,148.864
C01641=1233.179,-41.346,-38.683,-179.840,5.266,148.864
C01642=1233.174,-41.097,-38.695,-179.838,5.266,148.863
C01643=1233.168,-40.847,-38.709,-179.835,5.266,148.862
C01644=1233.164,-40.597,-38.722,-179.833,5.266,148.862
C01645=1233.159,-40.348,-38.734,-179.831,5.266,148.861
C01646=1233.153,-40.098,-38.747,-179.828,5.267,148.860
C01647=1233.148,-39.848,-38.760,-179.826,5.266,148.860
C01648=1233.143,-39.599,-38.773,-179.823,5.267,148.859
C01649=1233.139,-39.349,-38.786,-179.821,5.267,148.858
C01650=1233.133,-39.099,-38.799,-179.818,5.267,148.857
C01651=1233.128,-38.850,-38.812,-179.816,5.268,148.857
C01652=1233.123,-38.600,-38.825,-179.814,5.267,148.856
C01653=1233.117,-38.351,-38.839,-179.811,5.268,148.855
C01654=1233.112,-38.101,-38.851,-179.809,5.267,148.855
C01655=1233.108,-37.851,-38.864,-179.806,5.268,148.854
C01656=1233.102,-37.602,-38.877,-179.804,5.267,148.853
C01657=1233.097,-37.352,-38.890,-179.801,5.268,148.852
C01658=1233.092,-37.102,-38.903,-179.798,5.268,148.852
C01659=1233.086,-36.853,-38.916,-179.796,5.268,148.851
C01660=1233.082,-36.603,-38.930,-179.794,5.268,148.850
C01661=1233.077,-36.354,-38.942,-179.792,5.268,148.850
C01662=1233.071,-36.104,-38.956,-179.789,5.269,148.849
C01663=1233.067,-35.854,-38.969,-179.786,5.269,148.848
C01664=1233.062,-35.605,-38.981,-179.784,5.269,148.847
C01665=1233.056,-35.355,-38.995,-179.781,5.269,148.847
C01666=1233.052,-35.106,-39.008,-179.779,5.269,148.846
C01667=1233.046,-34.856,-39.022,-179.777,5.269,148.845
C01668=1233.041,-34.606,-39.034,-179.774,5.270,148.845
C01669=1233.036,-34.357,-39.047,-179.772,5.270,148.844
C01670=1233.031,-34.107,-39.060,-179.769,5.270,148.843
C01671=1233.026,-33.858,-39.074,-179.767,5.270,148.843
C01672=1233.021,-33.608,-39.087,-179.765,5.270,148.842
C01673=1233.016,-33.358,-39.100,-179.762,5.271,148.841
C01674=1233.011,-33.108,-39.113,-179.760,5.271,148.840
C01675=1233.005,-32.859,-39.127,-179.757,5.271,148.839
C01676=1233.000,-32.610,-39.139,-179.755,5.270,148.839
C01677=1232.995,-32.360,-39.153,-179.752,5.271,148.838
C01678=1232.990,-32.111,-39.166,-179.749,5.271,148.837
C01679=1232.985,-31.861,-39.180,-179.747,5.271,148.837
C01680=1232.980,-31.611,-39.192,-179.744,5.272,148.836
C01681=1232.976,-31.362,-39.206,-179.742,5.272,148.835
C01682=1232.970,-31.112,-39.219,-179.740,5.272,148.835
C01683=1232.965,-30.862,-39.232,-179.737,5.272,148.834
C01684=1232.959,-30.613,-39.245,-179.735,5.272,148.833
C01685=1232.955,-30.363,-39.259,-179.732,5.272,148.833
C01686=1232.949,-30.114,-39.272,-179.730,5.273,148.832
C01687=1232.945,-29.864,-39.286,-179.728,5.273,148.831
C01688=1232.939,-29.615,-39.299,-179.725,5.273,148.830
C01689=1232.935,-29.365,-39.312,-179.723,5.273,148.830
C01690=1232.929,-29.116,-39.326,-179.720,5.273,148.829
C01691=1232.925,-28.866,-39.339,-179.718,5.274,148.828
C01692=1232.919,-28.616,-39.352,-179.715,5.274,148.828
C01693=1232.915,-28.367,-39.366,-179.713,5.274,148.827
C01694=1232.909,-28.117,-39.379,-179.710,5.273,148.826
C01695=1232.904,-27.868,-39.393,-179.708,5.274,148.825
C01696=1232.899,-27.618,-39.406,-179.705,5.274,148.825
C01697=1232.894,-27.368,-39.420,-179.703,5.274,148.824
C01698=1232.889,-27.119,-39.433,-179.700,5.275,148.823
C01699=1232.883,-26.869,-39.446,-179.697,5.275,148.823
C01700=1232.878,-26.620,-39.460,-179.695,5.275,148.822
C01701=1232.873,-26.370,-39.473,-179.693,5.275,148.821
C01702=1232.868,-26.121,-39.487,-179.691,5.275,148.820
C01703=1232.863,-25.871,-39.500,-179.688,5.276,148.820
C01704=1232.859,-25.621,-39.514,-179.685,5.276,148.819
C01705=1232.853,-25.372,-39.527,-179.683,5.276,148.818
C01706=1232.848,-25.122,-39.541,-179.681,5.276,148.818
C01707=1232.843,-24.872,-39.554,-179.678,5.277,148.817
C01708=1232.838,-24.623,-39.568,-179.676,5.276,148.816
C01709=1232.833,-24.373,-39.581,-179.673,5.277,148.816
C01710=1232.828,-24.124,-39.595,-179.671,5.277,148.815
C01711=1232.823,-23.873,-39.609,-179.668,5.277,148.814
C01712=1232.818,-23.625,-39.622,-179.666,5.278,148.813
C01713=1232.813,-23.374,-39.635,-179.664,5.277,148.813
C01714=1232.808,-23.126,-39.649,-179.661,5.278,148.812
C01715=1232.803,-22.876,-39.663,-179.658,5.278,148.811
C01716=1232.797,-22.606,-39.677,-179.656,5.278,148.810
C01717=1232.791,-22.337,-39.692,-179.653,5.278,148.810
C01718=1232.786,-22.068,-39.706,-179.650,5.279,148.809
C01719=1232.781,-21.799,-39.721,-179.647,5.279,148.808
C01720=1232.776,-21.549,-39.736,-179.645,5.279,148.807
C01721=1232.770,-21.299,-39.749,-179.643,5.279,148.807
C01722=1232.766,-21.050,-39.762,-179.640,5.280,148.806
C01723=1232.760,-20.801,-39.776,-179.638,5.279,148.805
C01724=1232.755,-20.551,-39.790,-179.635,5.280,148.805
C01725=1232.751,-20.301,-39.804,-179.633,5.280,148.804
C01726=1232.745,-20.052,-39.817,-179.630,5.280,148.803
C01727=1232.740,-19.802,-39.831,-179.628,5.281,148.803
C01728=1232.735,-19.553,-39.844,-179.626,5.280,148.802
C01729=1232.730,-19.303,-39.858,-179.623,5.281,148.801
C01730=1232.725,-19.053,-39.872,-179.620,5.281,148.800
C01731=1232.719,-18.804,-39.886,-179.618,5.281,148.800
C01732=1232.715,-18.554,-39.899,-179.616,5.281,148.799
C01733=1232.710,-18.304,-39.913,-179.613,5.282,148.798
C01734=1232.704,-18.055,-39.927,-179.611,5.282,148.798
C01735=1232.699,-17.806,-39.942,-179.608,5.282,148.797
C01736=1232.695,-17.556,-39.955,-179.605,5.282,148.796
C01737=1232.689,-17.307,-39.969,-179.603,5.282,148.795
C01738=1232.684,-17.057,-39.983,-179.600,5.283,148.795
C01739=1232.679,-16.807,-39.997,-179.598,5.283,148.794
C01740=1232.674,-16.558,-40.010,-179.596,5.283,148.793
C01741=1232.669,-16.308,-40.024,-179.593,5.283,148.793
C01742=1232.664,-16.059,-40.038,-179.590,5.284,148.792
C01743=1232.659,-15.810,-40.052,-179.588,5.284,148.791
C01744=1232.654,-15.559,-40.066,-179.586,5.284,148.791
C01745=1232.649,-15.310,-40.079,-179.583,5.285,148.790
C01746=1232.644,-15.061,-40.093,-179.581,5.284,148.789
C01747=1232.639,-14.811,-40.108,-179.578,5.285,148.788
C01748=1232.634,-14.561,-40.122,-179.576,5.285,148.788
C01749=1232.629,-14.311,-40.135,-179.573,5.285,148.787
C01750=1232.624,-14.062,-40.149,-179.571,5.286,148.786
C01751=1232.619,-13.813,-40.163,-179.568,5.286,148.786
C01752=1232.614,-13.563,-40.177,-179.566,5.286,148.785
C01753=1232.608,-13.314,-40.191,-179.563,5.286,148.784
C01754=1232.603,-13.064,-40.205,-179.561,5.287,148.784
C01755=1232.599,-12.814,-40.220,-179.559,5.286,148.783
C01756=1232.593,-12.564,-40.233,-179.556,5.287,148.782
C01757=1232.588,-12.315,-40.247,-179.553,5.288,148.781
C01758=1232.583,-12.066,-40.261,-179.551,5.287,148.781
C01759=1232.579,-11.816,-40.275,-179.548,5.287,148.780
C01760=1232.574,-11.566,-40.289,-179.545,5.288,148.779
C01761=1232.568,-11.317,-40.303,-179.543,5.288,148.778
C01762=1232.563,-11.068,-40.318,-179.541,5.288,148.778
C01763=1232.558,-10.818,-40.332,-179.538,5.289,148.777
C01764=1232.553,-10.568,-40.346,-179.536,5.288,148.776
C01765=1232.548,-10.319,-40.360,-179.533,5.289,148.776
C01766=1232.543,-10.070,-40.374,-179.531,5.289,148.775
C01767=1232.538,-9.820,-40.388,-179.529,5.289,148.774
C01768=1232.533,-9.570,-40.402,-179.526,5.290,148.774
C01769=1232.528,-9.321,-40.416,-179.523,5.290,148.773
C01770=1232.523,-9.071,-40.430,-179.521,5.290,148.772
C01771=1232.518,-8.821,-40.444,-179.519,5.290,148.772
C01772=1232.513,-8.572,-40.458,-179.516,5.291,148.771
C01773=1232.508,-8.322,-40.473,-179.514,5.291,148.770
C01774=1232.502,-8.073,-40.487,-179.511,5.291,148.769
C01775=1232.497,-7.823,-40.501,-179.508,5.292,148.769
C01776=1232.492,-7.573,-40.515,-179.506,5.291,148.768
C01777=1232.488,-7.324,-40.530,-179.504,5.292,148.767
C01778=1232.483,-7.075,-40.544,-179.501,5.292,148.767
C01779=1232.478,-6.825,-40.559,-179.499,5.292,148.766
C01780=1232.472,-6.576,-40.573,-179.496,5.293,148.765
C01781=1232.467,-6.326,-40.587,-179.494,5.293,148.765
C01782=1232.462,-6.076,-40.601,-179.492,5.293,148.764
C01783=1232.457,-5.827,-40.615,-179.489,5.293,148.763
C01784=1232.452,-5.577,-40.630,-179.486,5.294,148.763
C01785=1232.447,-5.328,-40.644,-179.484,5.294,148.762
C01786=1232.442,-5.078,-40.658,-179.482,5.294,148.761
C01787=1232.437,-4.829,-40.672,-179.479,5.295,148.761
C01788=1232.432,-4.579,-40.686,-179.476,5.295,148.760
C01789=1232.427,-4.330,-40.701,-179.474,5.295,148.759
C01790=1232.422,-4.080,-40.716,-179.471,5.295,148.758
C01791=1232.417,-3.830,-40.730,-179.468,5.296,148.758
C01792=1232.412,-3.581,-40.744,-179.466,5.295,148.757
C01793=1232.407,-3.332,-40.758,-179.464,5.296,148.756
C01794=1232.402,-3.082,-40.772,-179.461,5.296,148.755
C01795=1232.397,-2.832,-40.787,-179.459,5.296,148.755
C01796=1232.392,-2.583,-40.802,-179.456,5.297,148.754
C01797=1232.387,-2.333,-40.816,-179.454,5.297,148.753
C01798=1232.382,-2.084,-40.830,-179.451,5.298,148.753
C01799=1232.377,-1.834,-40.845,-179.449,5.297,148.752
C01800=1232.372,-1.585,-40.858,-179.446,5.298,148.751
C01801=1232.367,-1.336,-40.874,-179.444,5.298,148.751
C01802=1232.362,-1.086,-40.888,-179.442,5.298,148.750
C01803=1232.357,-0.836,-40.903,-179.439,5.299,148.749
C01804=1232.352,-0.587,-40.917,-179.436,5.299,148.749
C01805=1232.347,-0.337,-40.932,-179.434,5.299,148.748
C01806=1232.342,-0.088,-40.946,-179.431,5.299,148.747
C01807=1232.337,0.162,-40.960,-179.429,5.300,148.746
C01808=1232.332,0.412,-40.975,-179.426,5.301,148.746
C01809=1232.327,0.661,-40.990,-179.424,5.300,148.745
C01810=1232.321,0.910,-41.004,-179.421,5.301,148.744
C01811=1232.316,1.160,-41.018,-179.419,5.301,148.744
C01812=1232.312,1.409,-41.033,-179.417,5.301,148.743
C01813=1232.307,1.659,-41.048,-179.414,5.302,148.742
C01814=1232.302,1.908,-41.062,-179.411,5.302,148.742
C01815=1232.296,2.158,-41.077,-179.409,5.303,148.741
C01816=1232.291,2.407,-41.092,-179.407,5.302,148.740
C01817=1232.286,2.657,-41.106,-179.404,5.303,148.740
C01818=1232.281,2.907,-41.120,-179.401,5.303,148.739
C01819=1232.277,3.156,-41.135,-179.399,5.303,148.738
C01820=1232.271,3.425,-41.152,-179.396,5.303,148.737
C01821=1232.266,3.694,-41.167,-179.393,5.304,148.737
C01822=1232.261,3.963,-41.183,-179.391,5.304,148.736
C01823=1232.256,4.231,-41.199,-179.388,5.305,148.735
C01824=1232.250,4.481,-41.214,-179.386,5.305,148.735
C01825=1232.245,4.731,-41.228,-179.383,5.305,148.734
